Yaskawa INFORM job: A_ROOF_SIDE_0617_2_PAINT_47.JBI

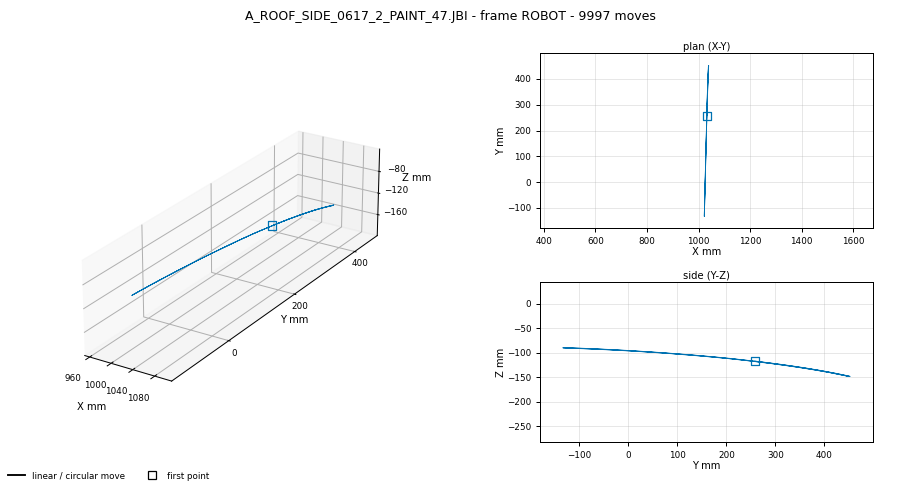
[picture p0: tool path of A_ROOF_SIDE_0617_2_PAINT_47.JBI in frame ROBOT, 9997 of 9997 moves have a stored position in this frame; points joined in program order, loops and branches not executed]
/JOB
//NAME A_ROOF_SIDE_0617_2_PAINT47
//POS
///NPOS 9997,0,0,0,0,0
///TOOL 1
///USER 0
///POSTYPE ROBOT
///RECTAN
///RCONF 1,0,0,0,0,0,0,0,0,0,0,0,0,0,0,0,0,0,0,0,0,0,0,0
C00000=1032.449,258.008,-117.083,170.684,44.569,158.533
C00001=1032.456,258.256,-117.113,170.687,44.569,158.534
C00002=1032.463,258.505,-117.142,170.690,44.569,158.534
C00003=1032.469,258.753,-117.172,170.693,44.568,158.534
C00004=1032.477,259.001,-117.201,170.697,44.568,158.535
C00005=1032.483,259.249,-117.230,170.701,44.568,158.535
C00006=1032.490,259.497,-117.260,170.704,44.568,158.535
C00007=1032.497,259.745,-117.290,170.707,44.567,158.535
C00008=1032.504,259.994,-117.319,170.711,44.567,158.536
C00009=1032.510,260.241,-117.349,170.714,44.567,158.536
C00010=1032.517,260.490,-117.379,170.718,44.567,158.536
C00011=1032.525,260.738,-117.408,170.721,44.567,158.537
C00012=1032.531,260.986,-117.437,170.725,44.566,158.537
C00013=1032.538,261.234,-117.467,170.728,44.566,158.537
C00014=1032.545,261.482,-117.497,170.731,44.566,158.537
C00015=1032.552,261.730,-117.527,170.734,44.566,158.538
C00016=1032.558,261.979,-117.556,170.739,44.566,158.538
C00017=1032.565,262.227,-117.586,170.742,44.566,158.538
C00018=1032.572,262.475,-117.617,170.745,44.566,158.539
C00019=1032.581,262.826,-117.659,170.749,44.566,158.539
C00020=1032.590,263.179,-117.701,170.755,44.566,158.540
C00021=1032.600,263.530,-117.744,170.759,44.566,158.540
C00022=1032.609,263.882,-117.786,170.765,44.566,158.541
C00023=1032.616,264.130,-117.817,170.768,44.566,158.541
C00024=1032.623,264.378,-117.846,170.771,44.566,158.541
C00025=1032.630,264.626,-117.876,170.775,44.566,158.541
C00026=1032.636,264.875,-117.907,170.779,44.566,158.542
C00027=1032.643,265.122,-117.937,170.782,44.566,158.542
C00028=1032.650,265.370,-117.967,170.786,44.566,158.542
C00029=1032.656,265.619,-117.997,170.789,44.566,158.543
C00030=1032.662,265.867,-118.027,170.792,44.566,158.543
C00031=1032.670,266.115,-118.057,170.796,44.565,158.543
C00032=1032.677,266.363,-118.087,170.800,44.565,158.544
C00033=1032.683,266.611,-118.117,170.803,44.565,158.544
C00034=1032.690,266.859,-118.148,170.806,44.565,158.544
C00035=1032.697,267.108,-118.178,170.810,44.565,158.545
C00036=1032.703,267.355,-118.208,170.814,44.565,158.545
C00037=1032.710,267.604,-118.238,170.817,44.565,158.545
C00038=1032.717,267.851,-118.269,170.821,44.566,158.546
C00039=1032.723,268.099,-118.299,170.824,44.566,158.546
C00040=1032.730,268.347,-118.329,170.828,44.565,158.546
C00041=1032.737,268.596,-118.360,170.831,44.565,158.547
C00042=1032.743,268.843,-118.390,170.835,44.565,158.547
C00043=1032.750,269.092,-118.421,170.838,44.565,158.547
C00044=1032.757,269.340,-118.451,170.842,44.566,158.548
C00045=1032.764,269.588,-118.481,170.846,44.566,158.548
C00046=1032.770,269.835,-118.512,170.849,44.566,158.549
C00047=1032.777,270.084,-118.542,170.852,44.566,158.549
C00048=1032.784,270.332,-118.573,170.856,44.566,158.549
C00049=1032.791,270.580,-118.603,170.860,44.566,158.549
C00050=1032.797,270.828,-118.634,170.864,44.566,158.550
C00051=1032.804,271.076,-118.664,170.867,44.566,158.550
C00052=1032.811,271.324,-118.695,170.870,44.566,158.551
C00053=1032.818,271.573,-118.725,170.874,44.566,158.551
C00054=1032.824,271.820,-118.756,170.878,44.567,158.551
C00055=1032.831,272.068,-118.786,170.881,44.566,158.552
C00056=1032.837,272.317,-118.817,170.885,44.566,158.552
C00057=1032.844,272.564,-118.848,170.889,44.567,158.553
C00058=1032.851,272.812,-118.878,170.892,44.567,158.553
C00059=1032.857,273.060,-118.909,170.896,44.567,158.553
C00060=1032.865,273.308,-118.940,170.900,44.567,158.554
C00061=1032.871,273.557,-118.970,170.903,44.567,158.554
C00062=1032.878,273.804,-119.002,170.907,44.567,158.554
C00063=1032.884,274.052,-119.031,170.910,44.568,158.555
C00064=1032.891,274.300,-119.063,170.914,44.568,158.555
C00065=1032.897,274.548,-119.094,170.918,44.568,158.555
C00066=1032.905,274.796,-119.124,170.921,44.568,158.556
C00067=1032.911,275.045,-119.155,170.926,44.568,158.556
C00068=1032.918,275.292,-119.187,170.929,44.568,158.557
C00069=1032.925,275.540,-119.216,170.932,44.569,158.557
C00070=1032.931,275.788,-119.248,170.936,44.569,158.557
C00071=1032.938,276.036,-119.279,170.940,44.569,158.558
C00072=1032.945,276.284,-119.309,170.943,44.569,158.558
C00073=1032.952,276.532,-119.341,170.947,44.569,158.558
C00074=1032.958,276.780,-119.372,170.951,44.569,158.559
C00075=1032.969,277.137,-119.415,170.957,44.569,158.560
C00076=1032.978,277.493,-119.460,170.961,44.570,158.560
C00077=1032.988,277.850,-119.505,170.967,44.570,158.561
C00078=1032.997,278.206,-119.549,170.972,44.570,158.561
C00079=1033.004,278.453,-119.581,170.976,44.571,158.562
C00080=1033.011,278.702,-119.612,170.980,44.571,158.562
C00081=1033.017,278.950,-119.643,170.984,44.571,158.562
C00082=1033.024,279.198,-119.674,170.987,44.571,158.563
C00083=1033.031,279.446,-119.706,170.992,44.572,158.563
C00084=1033.037,279.694,-119.737,170.995,44.572,158.564
C00085=1033.044,279.942,-119.768,170.998,44.572,158.564
C00086=1033.051,280.190,-119.799,171.003,44.573,158.565
C00087=1033.058,280.438,-119.830,171.006,44.573,158.565
C00088=1033.065,280.686,-119.862,171.010,44.573,158.565
C00089=1033.071,280.933,-119.893,171.014,44.573,158.566
C00090=1033.078,281.181,-119.925,171.018,44.574,158.566
C00091=1033.085,281.429,-119.956,171.021,44.574,158.567
C00092=1033.092,281.677,-119.987,171.025,44.574,158.567
C00093=1033.098,281.925,-120.019,171.029,44.575,158.568
C00094=1033.105,282.173,-120.050,171.032,44.575,158.568
C00095=1033.112,282.421,-120.082,171.037,44.575,158.568
C00096=1033.119,282.669,-120.113,171.040,44.576,158.569
C00097=1033.125,282.917,-120.145,171.045,44.575,158.569
C00098=1033.132,283.165,-120.176,171.048,44.576,158.570
C00099=1033.139,283.412,-120.207,171.052,44.577,158.570
C00100=1033.145,283.660,-120.239,171.056,44.576,158.570
C00101=1033.153,283.908,-120.270,171.059,44.577,158.571
C00102=1033.160,284.156,-120.301,171.064,44.577,158.571
C00103=1033.166,284.404,-120.333,171.067,44.578,158.572
C00104=1033.173,284.652,-120.364,171.071,44.578,158.572
C00105=1033.180,284.900,-120.395,171.075,44.578,158.573
C00106=1033.187,285.147,-120.427,171.079,44.579,158.573
C00107=1033.194,285.396,-120.459,171.083,44.579,158.574
C00108=1033.201,285.644,-120.490,171.087,44.579,158.574
C00109=1033.208,285.891,-120.522,171.091,44.580,158.575
C00110=1033.214,286.139,-120.554,171.094,44.580,158.575
C00111=1033.221,286.387,-120.585,171.098,44.580,158.575
C00112=1033.228,286.635,-120.617,171.102,44.581,158.576
C00113=1033.235,286.883,-120.648,171.106,44.581,158.576
C00114=1033.241,287.130,-120.681,171.111,44.582,158.577
C00115=1033.248,287.379,-120.713,171.114,44.582,158.577
C00116=1033.255,287.627,-120.744,171.118,44.582,158.578
C00117=1033.262,287.874,-120.776,171.122,44.583,158.578
C00118=1033.269,288.122,-120.808,171.125,44.583,158.579
C00119=1033.275,288.370,-120.839,171.130,44.584,158.579
C00120=1033.282,288.618,-120.872,171.133,44.584,158.580
C00121=1033.289,288.866,-120.904,171.138,44.585,158.580
C00122=1033.296,289.114,-120.936,171.142,44.585,158.581
C00123=1033.303,289.361,-120.967,171.146,44.585,158.581
C00124=1033.310,289.609,-120.999,171.150,44.586,158.582
C00125=1033.316,289.857,-121.031,171.154,44.586,158.582
C00126=1033.322,290.105,-121.063,171.157,44.586,158.582
C00127=1033.330,290.353,-121.095,171.162,44.587,158.583
C00128=1033.337,290.601,-121.127,171.165,44.587,158.583
C00129=1033.343,290.848,-121.159,171.170,44.588,158.584
C00130=1033.350,291.096,-121.192,171.174,44.588,158.584
C00131=1033.361,291.464,-121.239,171.179,44.589,158.585
C00132=1033.371,291.833,-121.287,171.185,44.590,158.586
C00133=1033.381,292.202,-121.335,171.192,44.591,158.587
C00134=1033.391,292.570,-121.383,171.198,44.591,158.587
C00135=1033.398,292.818,-121.414,171.201,44.592,158.588
C00136=1033.405,293.066,-121.447,171.206,44.592,158.588
C00137=1033.412,293.314,-121.479,171.209,44.593,158.589
C00138=1033.418,293.561,-121.511,171.214,44.593,158.589
C00139=1033.425,293.810,-121.544,171.218,44.595,158.590
C00140=1033.432,294.057,-121.576,171.222,44.595,158.590
C00141=1033.439,294.304,-121.608,171.226,44.596,158.591
C00142=1033.446,294.553,-121.641,171.230,44.596,158.591
C00143=1033.453,294.801,-121.673,171.234,44.596,158.592
C00144=1033.459,295.048,-121.705,171.238,44.597,158.592
C00145=1033.466,295.296,-121.738,171.242,44.598,158.593
C00146=1033.473,295.544,-121.771,171.247,44.598,158.594
C00147=1033.479,295.791,-121.803,171.250,44.599,158.594
C00148=1033.486,296.039,-121.836,171.255,44.599,158.595
C00149=1033.493,296.287,-121.869,171.258,44.601,158.595
C00150=1033.500,296.534,-121.901,171.263,44.601,158.596
C00151=1033.506,296.782,-121.934,171.267,44.601,158.596
C00152=1033.513,297.030,-121.967,171.271,44.603,158.597
C00153=1033.520,297.278,-121.999,171.276,44.603,158.597
C00154=1033.526,297.525,-122.032,171.279,44.604,158.598
C00155=1033.533,297.774,-122.065,171.284,44.605,158.599
C00156=1033.540,298.021,-122.097,171.288,44.605,158.599
C00157=1033.546,298.268,-122.130,171.292,44.606,158.600
C00158=1033.553,298.517,-122.163,171.296,44.607,158.600
C00159=1033.560,298.764,-122.197,171.300,44.607,158.601
C00160=1033.568,299.012,-122.229,171.304,44.608,158.601
C00161=1033.574,299.259,-122.262,171.309,44.609,158.602
C00162=1033.580,299.507,-122.295,171.313,44.609,158.602
C00163=1033.587,299.755,-122.328,171.317,44.610,158.603
C00164=1033.594,300.002,-122.360,171.322,44.611,158.603
C00165=1033.601,300.250,-122.394,171.325,44.612,158.604
C00166=1033.608,300.498,-122.427,171.330,44.612,158.605
C00167=1033.615,300.746,-122.459,171.334,44.613,158.605
C00168=1033.621,300.993,-122.492,171.338,44.614,158.606
C00169=1033.629,301.241,-122.526,171.343,44.614,158.606
C00170=1033.635,301.489,-122.558,171.347,44.615,158.607
C00171=1033.643,301.737,-122.591,171.351,44.616,158.607
C00172=1033.649,301.983,-122.624,171.356,44.617,158.608
C00173=1033.656,302.232,-122.657,171.359,44.617,158.609
C00174=1033.662,302.479,-122.690,171.364,44.618,158.609
C00175=1033.670,302.727,-122.723,171.368,44.619,158.610
C00176=1033.677,302.974,-122.756,171.373,44.620,158.610
C00177=1033.684,303.223,-122.789,171.377,44.620,158.611
C00178=1033.690,303.470,-122.823,171.381,44.622,158.612
C00179=1033.698,303.718,-122.855,171.385,44.622,158.612
C00180=1033.705,303.965,-122.889,171.390,44.623,158.613
C00181=1033.711,304.213,-122.922,171.394,44.623,158.613
C00182=1033.718,304.461,-122.956,171.399,44.624,158.614
C00183=1033.725,304.708,-122.988,171.403,44.625,158.614
C00184=1033.733,304.955,-123.022,171.407,44.626,158.615
C00185=1033.740,305.204,-123.055,171.412,44.627,158.616
C00186=1033.746,305.451,-123.088,171.416,44.627,158.616
C00187=1033.757,305.836,-123.139,171.422,44.629,158.617
C00188=1033.768,306.222,-123.192,171.429,44.630,158.618
C00189=1033.779,306.608,-123.243,171.436,44.631,158.619
C00190=1033.791,306.993,-123.295,171.443,44.632,158.620
C00191=1033.798,307.241,-123.328,171.448,44.633,158.621
C00192=1033.804,307.488,-123.362,171.452,44.634,158.621
C00193=1033.811,307.736,-123.395,171.456,44.635,158.622
C00194=1033.818,307.984,-123.428,171.461,44.636,158.623
C00195=1033.826,308.231,-123.462,171.465,44.637,158.623
C00196=1033.833,308.478,-123.495,171.470,44.638,158.624
C00197=1033.840,308.726,-123.529,171.474,44.638,158.624
C00198=1033.847,308.974,-123.562,171.479,44.639,158.625
C00199=1033.855,309.222,-123.595,171.483,44.641,158.626
C00200=1033.861,309.469,-123.629,171.487,44.641,158.626
C00201=1033.869,309.716,-123.663,171.492,44.642,158.627
C00202=1033.876,309.964,-123.696,171.497,44.643,158.628
C00203=1033.883,310.212,-123.730,171.502,44.644,158.628
C00204=1033.891,310.460,-123.763,171.505,44.644,158.629
C00205=1033.898,310.707,-123.797,171.510,44.645,158.629
C00206=1033.904,310.954,-123.830,171.515,44.646,158.630
C00207=1033.912,311.202,-123.864,171.520,44.647,158.631
C00208=1033.919,311.450,-123.898,171.524,44.648,158.631
C00209=1033.926,311.697,-123.932,171.528,44.650,158.632
C00210=1033.933,311.945,-123.965,171.533,44.651,158.633
C00211=1033.939,312.192,-123.999,171.538,44.651,158.633
C00212=1033.946,312.440,-124.033,171.542,44.653,158.634
C00213=1033.953,312.688,-124.067,171.546,44.654,158.635
C00214=1033.960,312.935,-124.102,171.551,44.655,158.635
C00215=1033.967,313.183,-124.136,171.556,44.656,158.636
C00216=1033.973,313.430,-124.170,171.560,44.657,158.637
C00217=1033.981,313.678,-124.204,171.565,44.658,158.637
C00218=1033.988,313.925,-124.238,171.569,44.659,158.638
C00219=1033.994,314.173,-124.273,171.574,44.660,158.639
C00220=1034.002,314.420,-124.307,171.579,44.661,158.640
C00221=1034.008,314.668,-124.341,171.583,44.663,158.640
C00222=1034.016,314.915,-124.376,171.588,44.663,158.641
C00223=1034.022,315.162,-124.409,171.593,44.664,158.642
C00224=1034.029,315.410,-124.444,171.597,44.665,158.642
C00225=1034.036,315.657,-124.478,171.602,44.667,158.643
C00226=1034.043,315.905,-124.512,171.606,44.668,158.644
C00227=1034.050,316.152,-124.547,171.611,44.669,158.645
C00228=1034.057,316.400,-124.581,171.616,44.670,158.645
C00229=1034.064,316.648,-124.615,171.621,44.671,158.646
C00230=1034.071,316.895,-124.650,171.626,44.673,158.647
C00231=1034.078,317.143,-124.684,171.629,44.674,158.647
C00232=1034.085,317.390,-124.719,171.634,44.675,158.648
C00233=1034.092,317.638,-124.753,171.639,44.676,158.649
C00234=1034.099,317.885,-124.788,171.644,44.677,158.650
C00235=1034.106,318.133,-124.822,171.649,44.678,158.650
C00236=1034.113,318.380,-124.857,171.654,44.679,158.651
C00237=1034.120,318.628,-124.890,171.659,44.681,158.652
C00238=1034.127,318.875,-124.926,171.662,44.682,158.652
C00239=1034.135,319.122,-124.960,171.667,44.683,158.653
C00240=1034.141,319.370,-124.995,171.672,44.685,158.654
C00241=1034.149,319.617,-125.029,171.677,44.686,158.655
C00242=1034.157,319.866,-125.063,171.682,44.687,158.655
C00243=1034.167,320.256,-125.118,171.689,44.689,158.657
C00244=1034.179,320.646,-125.173,171.697,44.691,158.658
C00245=1034.189,321.036,-125.227,171.705,44.692,158.659
C00246=1034.201,321.427,-125.282,171.713,44.695,158.660
C00247=1034.209,321.674,-125.317,171.717,44.696,158.661
C00248=1034.215,321.922,-125.351,171.722,44.697,158.662
C00249=1034.223,322.169,-125.386,171.727,44.698,158.662
C00250=1034.230,322.417,-125.421,171.731,44.700,158.663
C00251=1034.238,322.664,-125.456,171.736,44.701,158.664
C00252=1034.244,322.911,-125.491,171.741,44.702,158.665
C00253=1034.252,323.158,-125.525,171.746,44.703,158.665
C00254=1034.259,323.407,-125.560,171.751,44.705,158.666
C00255=1034.266,323.654,-125.595,171.756,44.706,158.667
C00256=1034.273,323.901,-125.630,171.761,44.707,158.668
C00257=1034.281,324.149,-125.665,171.766,44.708,158.669
C00258=1034.288,324.396,-125.700,171.771,44.710,158.669
C00259=1034.296,324.643,-125.735,171.775,44.711,158.670
C00260=1034.303,324.892,-125.770,171.780,44.712,158.671
C00261=1034.310,325.139,-125.805,171.785,44.714,158.672
C00262=1034.317,325.386,-125.840,171.790,44.715,158.672
C00263=1034.325,325.634,-125.875,171.795,44.717,158.673
C00264=1034.332,325.881,-125.910,171.800,44.718,158.674
C00265=1034.340,326.128,-125.944,171.805,44.719,158.675
C00266=1034.347,326.376,-125.980,171.810,44.721,158.676
C00267=1034.354,326.623,-126.014,171.815,44.722,158.676
C00268=1034.362,326.870,-126.050,171.820,44.723,158.677
C00269=1034.370,327.118,-126.085,171.826,44.724,158.678
C00270=1034.376,327.365,-126.120,171.831,44.726,158.679
C00271=1034.385,327.613,-126.155,171.836,44.727,158.680
C00272=1034.391,327.860,-126.190,171.841,44.729,158.681
C00273=1034.399,328.108,-126.225,171.846,44.730,158.681
C00274=1034.406,328.355,-126.261,171.851,44.732,158.682
C00275=1034.414,328.603,-126.297,171.856,44.733,158.683
C00276=1034.421,328.850,-126.332,171.861,44.734,158.684
C00277=1034.428,329.097,-126.367,171.866,44.736,158.685
C00278=1034.436,329.345,-126.402,171.871,44.737,158.686
C00279=1034.443,329.591,-126.438,171.876,44.739,158.686
C00280=1034.450,329.839,-126.474,171.881,44.740,158.687
C00281=1034.457,330.086,-126.510,171.886,44.742,158.688
C00282=1034.465,330.334,-126.545,171.891,44.744,158.689
C00283=1034.472,330.581,-126.581,171.896,44.745,158.690
C00284=1034.479,330.829,-126.616,171.901,44.747,158.691
C00285=1034.486,331.076,-126.652,171.906,44.748,158.691
C00286=1034.494,331.324,-126.688,171.912,44.750,158.692
C00287=1034.501,331.571,-126.724,171.917,44.751,158.693
C00288=1034.508,331.818,-126.760,171.922,44.753,158.694
C00289=1034.515,332.065,-126.795,171.928,44.755,158.695
C00290=1034.524,332.313,-126.831,171.933,44.756,158.696
C00291=1034.530,332.560,-126.866,171.938,44.758,158.697
C00292=1034.538,332.807,-126.902,171.943,44.759,158.698
C00293=1034.546,333.055,-126.938,171.948,44.761,158.699
C00294=1034.553,333.302,-126.974,171.954,44.762,158.699
C00295=1034.560,333.550,-127.010,171.959,44.764,158.700
C00296=1034.567,333.796,-127.045,171.964,44.766,158.701
C00297=1034.575,334.044,-127.082,171.969,44.768,158.702
C00298=1034.583,334.291,-127.118,171.974,44.769,158.703
C00299=1034.594,334.678,-127.174,171.983,44.772,158.705
C00300=1034.605,335.063,-127.230,171.991,44.774,158.706
C00301=1034.617,335.448,-127.286,172.000,44.777,158.707
C00302=1034.628,335.834,-127.343,172.008,44.780,158.709
C00303=1034.635,336.082,-127.380,172.013,44.781,158.710
C00304=1034.642,336.329,-127.415,172.018,44.783,158.711
C00305=1034.650,336.576,-127.452,172.024,44.785,158.712
C00306=1034.658,336.823,-127.488,172.029,44.786,158.712
C00307=1034.665,337.070,-127.524,172.034,44.788,158.713
C00308=1034.672,337.318,-127.561,172.039,44.790,158.714
C00309=1034.679,337.565,-127.597,172.045,44.792,158.715
C00310=1034.687,337.813,-127.633,172.051,44.793,158.716
C00311=1034.695,338.060,-127.670,172.056,44.796,158.717
C00312=1034.702,338.306,-127.706,172.061,44.797,158.718
C00313=1034.709,338.554,-127.743,172.066,44.799,158.719
C00314=1034.717,338.802,-127.779,172.073,44.801,158.720
C00315=1034.724,339.049,-127.815,172.078,44.803,158.721
C00316=1034.732,339.296,-127.852,172.083,44.804,158.722
C00317=1034.740,339.543,-127.888,172.088,44.806,158.723
C00318=1034.746,339.790,-127.925,172.095,44.808,158.724
C00319=1034.754,340.037,-127.962,172.100,44.810,158.725
C00320=1034.762,340.285,-127.998,172.105,44.812,158.726
C00321=1034.770,340.532,-128.034,172.111,44.813,158.727
C00322=1034.778,340.779,-128.071,172.116,44.815,158.728
C00323=1034.785,341.027,-128.108,172.122,44.818,158.729
C00324=1034.793,341.273,-128.145,172.127,44.820,158.730
C00325=1034.799,341.521,-128.181,172.133,44.821,158.731
C00326=1034.807,341.767,-128.218,172.138,44.823,158.732
C00327=1034.815,342.015,-128.254,172.144,44.825,158.733
C00328=1034.822,342.262,-128.292,172.150,44.827,158.734
C00329=1034.830,342.509,-128.328,172.155,44.829,158.735
C00330=1034.837,342.756,-128.366,172.160,44.831,158.736
C00331=1034.845,343.003,-128.402,172.167,44.833,158.737
C00332=1034.852,343.251,-128.439,172.172,44.835,158.738
C00333=1034.860,343.498,-128.476,172.177,44.837,158.739
C00334=1034.867,343.745,-128.514,172.184,44.839,158.740
C00335=1034.875,343.992,-128.550,172.189,44.841,158.741
C00336=1034.882,344.240,-128.587,172.194,44.843,158.742
C00337=1034.890,344.486,-128.624,172.200,44.845,158.743
C00338=1034.897,344.734,-128.662,172.206,44.847,158.744
C00339=1034.905,344.981,-128.698,172.211,44.849,158.745
C00340=1034.912,345.228,-128.736,172.217,44.851,158.746
C00341=1034.920,345.475,-128.773,172.223,44.853,158.747
C00342=1034.927,345.722,-128.810,172.228,44.855,158.748
C00343=1034.935,345.969,-128.847,172.234,44.857,158.749
C00344=1034.942,346.216,-128.885,172.240,44.859,158.750
C00345=1034.951,346.464,-128.922,172.246,44.861,158.752
C00346=1034.958,346.711,-128.959,172.251,44.863,158.753
C00347=1034.966,346.958,-128.997,172.257,44.866,158.754
C00348=1034.974,347.205,-129.034,172.263,44.867,158.755
C00349=1034.981,347.452,-129.071,172.269,44.870,158.756
C00350=1034.989,347.699,-129.108,172.275,44.872,158.757
C00351=1034.997,347.946,-129.146,172.280,44.874,158.758
C00352=1035.005,348.193,-129.183,172.287,44.876,158.759
C00353=1035.012,348.440,-129.221,172.292,44.878,158.760
C00354=1035.019,348.688,-129.258,172.298,44.881,158.761
C00355=1035.032,349.070,-129.316,172.308,44.884,158.763
C00356=1035.043,349.452,-129.375,172.316,44.887,158.765
C00357=1035.055,349.835,-129.432,172.325,44.891,158.766
C00358=1035.067,350.217,-129.491,172.334,44.894,158.768
C00359=1035.075,350.464,-129.529,172.341,44.896,158.769
C00360=1035.082,350.711,-129.566,172.346,44.899,158.771
C00361=1035.090,350.957,-129.604,172.352,44.901,158.772
C00362=1035.098,351.205,-129.642,172.358,44.904,158.773
C00363=1035.105,351.452,-129.680,172.364,44.905,158.774
C00364=1035.113,351.699,-129.718,172.370,44.908,158.775
C00365=1035.121,351.946,-129.756,172.376,44.910,158.776
C00366=1035.128,352.193,-129.794,172.382,44.913,158.777
C00367=1035.136,352.440,-129.832,172.388,44.915,158.778
C00368=1035.144,352.687,-129.869,172.395,44.917,158.780
C00369=1035.152,352.934,-129.908,172.400,44.920,158.781
C00370=1035.159,353.180,-129.946,172.407,44.922,158.782
C00371=1035.167,353.428,-129.984,172.412,44.924,158.783
C00372=1035.175,353.675,-130.022,172.419,44.926,158.784
C00373=1035.184,353.922,-130.060,172.424,44.929,158.785
C00374=1035.191,354.169,-130.098,172.431,44.931,158.787
C00375=1035.199,354.416,-130.136,172.437,44.934,158.788
C00376=1035.207,354.663,-130.174,172.443,44.936,158.789
C00377=1035.214,354.910,-130.212,172.449,44.938,158.790
C00378=1035.222,355.157,-130.251,172.455,44.941,158.791
C00379=1035.230,355.404,-130.289,172.461,44.944,158.793
C00380=1035.238,355.650,-130.327,172.468,44.945,158.794
C00381=1035.247,355.898,-130.365,172.473,44.948,158.795
C00382=1035.254,356.144,-130.404,172.480,44.951,158.796
C00383=1035.262,356.391,-130.442,172.487,44.953,158.798
C00384=1035.270,356.638,-130.481,172.492,44.956,158.799
C00385=1035.277,356.885,-130.520,172.499,44.958,158.800
C00386=1035.285,357.132,-130.558,172.505,44.961,158.801
C00387=1035.293,357.379,-130.597,172.511,44.963,158.802
C00388=1035.301,357.626,-130.635,172.518,44.966,158.804
C00389=1035.309,357.873,-130.673,172.524,44.968,158.805
C00390=1035.317,358.120,-130.712,172.530,44.971,158.806
C00391=1035.324,358.366,-130.750,172.536,44.973,158.807
C00392=1035.333,358.614,-130.789,172.543,44.976,158.809
C00393=1035.341,358.861,-130.828,172.549,44.978,158.810
C00394=1035.349,359.107,-130.867,172.555,44.981,158.811
C00395=1035.357,359.354,-130.905,172.562,44.983,158.812
C00396=1035.365,359.601,-130.944,172.569,44.986,158.814
C00397=1035.372,359.848,-130.982,172.574,44.989,158.815
C00398=1035.381,360.094,-131.021,172.581,44.992,158.816
C00399=1035.389,360.342,-131.060,172.587,44.994,158.818
C00400=1035.396,360.588,-131.099,172.594,44.997,158.819
C00401=1035.404,360.835,-131.138,172.600,45.000,158.820
C00402=1035.412,361.082,-131.177,172.606,45.002,158.821
C00403=1035.421,361.329,-131.216,172.613,45.005,158.823
C00404=1035.428,361.575,-131.254,172.620,45.008,158.824
C00405=1035.436,361.822,-131.294,172.627,45.010,158.825
C00406=1035.444,362.069,-131.333,172.632,45.013,158.827
C00407=1035.453,362.316,-131.372,172.639,45.016,158.828
C00408=1035.460,362.563,-131.412,172.646,45.019,158.830
C00409=1035.468,362.809,-131.450,172.652,45.021,158.831
C00410=1035.476,363.056,-131.490,172.659,45.024,158.832
C00411=1035.488,363.445,-131.552,172.669,45.029,158.834
C00412=1035.502,363.833,-131.614,172.680,45.033,158.836
C00413=1035.514,364.222,-131.675,172.690,45.038,158.839
C00414=1035.527,364.610,-131.738,172.700,45.042,158.841
C00415=1035.534,364.857,-131.778,172.707,45.045,158.842
C00416=1035.543,365.104,-131.816,172.714,45.048,158.844
C00417=1035.551,365.351,-131.856,172.721,45.050,158.845
C00418=1035.559,365.597,-131.895,172.728,45.053,158.846
C00419=1035.567,365.844,-131.935,172.734,45.056,158.848
C00420=1035.575,366.091,-131.975,172.741,45.059,158.849
C00421=1035.583,366.338,-132.014,172.747,45.062,158.850
C00422=1035.592,366.584,-132.053,172.754,45.065,158.852
C00423=1035.600,366.831,-132.093,172.761,45.068,158.853
C00424=1035.608,367.078,-132.133,172.768,45.071,158.855
C00425=1035.616,367.324,-132.173,172.774,45.074,158.856
C00426=1035.625,367.570,-132.213,172.781,45.077,158.858
C00427=1035.633,367.817,-132.252,172.788,45.080,158.859
C00428=1035.641,368.064,-132.292,172.795,45.083,158.860
C00429=1035.649,368.311,-132.331,172.802,45.086,158.862
C00430=1035.658,368.558,-132.372,172.809,45.089,158.863
C00431=1035.666,368.804,-132.411,172.816,45.092,158.865
C00432=1035.675,369.051,-132.451,172.823,45.095,158.866
C00433=1035.682,369.298,-132.491,172.829,45.098,158.868
C00434=1035.691,369.544,-132.531,172.836,45.101,158.869
C00435=1035.699,369.791,-132.571,172.843,45.104,158.870
C00436=1035.708,370.037,-132.611,172.850,45.107,158.872
C00437=1035.716,370.284,-132.651,172.857,45.110,158.873
C00438=1035.724,370.530,-132.692,172.864,45.113,158.875
C00439=1035.732,370.777,-132.732,172.872,45.116,158.876
C00440=1035.741,371.023,-132.772,172.879,45.119,158.878
C00441=1035.748,371.270,-132.811,172.886,45.123,158.880
C00442=1035.757,371.517,-132.853,172.893,45.126,158.881
C00443=1035.765,371.763,-132.893,172.900,45.129,158.882
C00444=1035.773,372.010,-132.932,172.907,45.132,158.884
C00445=1035.781,372.256,-132.973,172.914,45.135,158.885
C00446=1035.790,372.503,-133.014,172.921,45.139,158.887
C00447=1035.798,372.750,-133.055,172.928,45.142,158.889
C00448=1035.807,372.996,-133.095,172.935,45.145,158.890
C00449=1035.815,373.243,-133.135,172.943,45.148,158.892
C00450=1035.823,373.489,-133.176,172.950,45.152,158.893
C00451=1035.831,373.736,-133.216,172.957,45.155,158.895
C00452=1035.841,373.982,-133.257,172.964,45.158,158.896
C00453=1035.849,374.229,-133.297,172.971,45.162,158.898
C00454=1035.857,374.476,-133.338,172.978,45.165,158.899
C00455=1035.865,374.722,-133.379,172.986,45.168,158.901
C00456=1035.874,374.968,-133.419,172.994,45.172,158.903
C00457=1035.883,375.215,-133.460,173.001,45.175,158.904
C00458=1035.891,375.461,-133.501,173.008,45.178,158.906
C00459=1035.899,375.708,-133.542,173.015,45.182,158.907
C00460=1035.908,375.954,-133.582,173.023,45.185,158.909
C00461=1035.917,376.201,-133.623,173.030,45.188,158.911
C00462=1035.925,376.447,-133.664,173.037,45.192,158.912
C00463=1035.934,376.694,-133.705,173.045,45.195,158.914
C00464=1035.942,376.940,-133.746,173.052,45.198,158.915
C00465=1035.951,377.187,-133.786,173.060,45.202,158.917
C00466=1035.960,377.433,-133.828,173.067,45.205,158.919
C00467=1035.974,377.842,-133.895,173.079,45.211,158.921
C00468=1035.988,378.251,-133.964,173.092,45.217,158.924
C00469=1036.002,378.660,-134.032,173.105,45.223,158.927
C00470=1036.016,379.069,-134.100,173.117,45.229,158.930
C00471=1036.025,379.315,-134.142,173.125,45.232,158.931
C00472=1036.033,379.562,-134.183,173.132,45.236,158.933
C00473=1036.041,379.808,-134.225,173.140,45.239,158.935
C00474=1036.050,380.055,-134.267,173.147,45.243,158.937
C00475=1036.059,380.300,-134.308,173.156,45.247,158.938
C00476=1036.067,380.547,-134.349,173.163,45.250,158.940
C00477=1036.076,380.794,-134.391,173.170,45.254,158.942
C00478=1036.085,381.040,-134.433,173.178,45.257,158.943
C00479=1036.094,381.286,-134.474,173.186,45.262,158.945
C00480=1036.102,381.532,-134.516,173.194,45.265,158.947
C00481=1036.111,381.779,-134.558,173.202,45.269,158.949
C00482=1036.119,382.026,-134.599,173.210,45.272,158.950
C00483=1036.128,382.272,-134.641,173.217,45.276,158.952
C00484=1036.137,382.518,-134.682,173.224,45.280,158.954
C00485=1036.146,382.764,-134.724,173.233,45.284,158.956
C00486=1036.154,383.010,-134.766,173.240,45.287,158.957
C00487=1036.164,383.256,-134.808,173.248,45.291,158.959
C00488=1036.173,383.503,-134.850,173.257,45.295,158.961
C00489=1036.181,383.749,-134.892,173.264,45.298,158.963
C00490=1036.190,383.996,-134.934,173.273,45.302,158.964
C00491=1036.199,384.242,-134.975,173.280,45.306,158.966
C00492=1036.208,384.488,-135.017,173.289,45.310,158.968
C00493=1036.217,384.734,-135.060,173.296,45.314,158.970
C00494=1036.226,384.980,-135.101,173.304,45.317,158.972
C00495=1036.235,385.227,-135.143,173.312,45.322,158.973
C00496=1036.243,385.473,-135.186,173.320,45.325,158.975
C00497=1036.252,385.719,-135.228,173.329,45.329,158.977
C00498=1036.261,385.966,-135.269,173.336,45.333,158.979
C00499=1036.270,386.211,-135.312,173.345,45.337,158.981
C00500=1036.279,386.458,-135.354,173.353,45.341,158.983
C00501=1036.289,386.703,-135.396,173.360,45.345,158.985
C00502=1036.297,386.950,-135.438,173.369,45.349,158.986
C00503=1036.306,387.196,-135.481,173.377,45.353,158.988
C00504=1036.315,387.443,-135.523,173.385,45.357,158.990
C00505=1036.325,387.689,-135.565,173.394,45.361,158.992
C00506=1036.333,387.935,-135.608,173.402,45.365,158.994
C00507=1036.342,388.181,-135.650,173.410,45.369,158.996
C00508=1036.351,388.427,-135.692,173.418,45.373,158.998
C00509=1036.360,388.673,-135.736,173.427,45.377,159.000
C00510=1036.370,388.919,-135.778,173.435,45.381,159.002
C00511=1036.378,389.165,-135.821,173.443,45.386,159.004
C00512=1036.387,389.411,-135.864,173.452,45.389,159.006
C00513=1036.396,389.657,-135.907,173.460,45.394,159.008
C00514=1036.406,389.904,-135.950,173.469,45.398,159.009
C00515=1036.415,390.149,-135.992,173.478,45.402,159.012
C00516=1036.424,390.395,-136.035,173.485,45.406,159.013
C00517=1036.433,390.642,-136.078,173.494,45.410,159.015
C00518=1036.442,390.888,-136.121,173.503,45.415,159.017
C00519=1036.451,391.134,-136.163,173.511,45.419,159.019
C00520=1036.460,391.380,-136.207,173.520,45.423,159.021
C00521=1036.469,391.626,-136.250,173.529,45.427,159.023
C00522=1036.478,391.872,-136.293,173.536,45.432,159.025
C00523=1036.489,392.155,-136.342,173.546,45.437,159.028
C00524=1036.499,392.436,-136.392,173.556,45.441,159.030
C00525=1036.509,392.719,-136.441,173.567,45.447,159.032
C00526=1036.521,393.001,-136.491,173.576,45.452,159.035
C00527=1036.530,393.246,-136.535,173.585,45.456,159.037
C00528=1036.539,393.493,-136.578,173.593,45.460,159.039
C00529=1036.548,393.738,-136.621,173.602,45.465,159.041
C00530=1036.557,393.985,-136.665,173.611,45.469,159.043
C00531=1036.573,394.392,-136.737,173.626,45.476,159.046
C00532=1036.588,394.800,-136.808,173.640,45.484,159.050
C00533=1036.604,395.207,-136.881,173.655,45.491,159.053
C00534=1036.619,395.614,-136.953,173.670,45.499,159.057
C00535=1036.629,395.860,-136.997,173.679,45.503,159.059
C00536=1036.638,396.106,-137.041,173.688,45.508,159.061
C00537=1036.647,396.352,-137.085,173.697,45.512,159.063
C00538=1036.657,396.597,-137.128,173.706,45.517,159.066
C00539=1036.666,396.844,-137.172,173.715,45.521,159.068
C00540=1036.675,397.089,-137.216,173.724,45.526,159.070
C00541=1036.685,397.335,-137.260,173.733,45.530,159.072
C00542=1036.694,397.581,-137.304,173.742,45.535,159.074
C00543=1036.704,397.827,-137.348,173.751,45.540,159.076
C00544=1036.714,398.073,-137.392,173.760,45.544,159.079
C00545=1036.722,398.319,-137.436,173.769,45.549,159.081
C00546=1036.732,398.564,-137.480,173.779,45.554,159.083
C00547=1036.741,398.810,-137.524,173.788,45.558,159.085
C00548=1036.752,399.056,-137.568,173.797,45.563,159.087
C00549=1036.761,399.302,-137.612,173.806,45.568,159.090
C00550=1036.771,399.548,-137.657,173.816,45.573,159.092
C00551=1036.780,399.794,-137.701,173.826,45.577,159.094
C00552=1036.790,400.039,-137.746,173.835,45.582,159.097
C00553=1036.799,400.286,-137.790,173.844,45.587,159.099
C00554=1036.809,400.531,-137.835,173.854,45.592,159.101
C00555=1036.818,400.777,-137.879,173.863,45.597,159.103
C00556=1036.828,401.023,-137.924,173.872,45.602,159.106
C00557=1036.837,401.269,-137.968,173.882,45.606,159.108
C00558=1036.847,401.514,-138.013,173.891,45.612,159.110
C00559=1036.857,401.760,-138.057,173.901,45.616,159.113
C00560=1036.867,402.005,-138.102,173.911,45.621,159.115
C00561=1036.876,402.252,-138.146,173.920,45.626,159.117
C00562=1036.886,402.497,-138.191,173.930,45.631,159.120
C00563=1036.896,402.743,-138.236,173.939,45.636,159.122
C00564=1036.906,402.989,-138.281,173.949,45.641,159.124
C00565=1036.916,403.234,-138.326,173.959,45.646,159.127
C00566=1036.924,403.480,-138.372,173.968,45.651,159.129
C00567=1036.934,403.726,-138.416,173.978,45.656,159.132
C00568=1036.945,403.972,-138.462,173.988,45.661,159.134
C00569=1036.954,404.217,-138.506,173.998,45.666,159.136
C00570=1036.964,404.463,-138.551,174.007,45.672,159.139
C00571=1036.973,404.708,-138.597,174.018,45.677,159.141
C00572=1036.984,404.954,-138.642,174.027,45.682,159.144
C00573=1036.993,405.200,-138.687,174.037,45.687,159.146
C00574=1037.003,405.445,-138.733,174.047,45.692,159.149
C00575=1037.013,405.691,-138.779,174.057,45.697,159.151
C00576=1037.023,405.937,-138.823,174.066,45.703,159.154
C00577=1037.033,406.182,-138.869,174.077,45.708,159.156
C00578=1037.043,406.428,-138.914,174.087,45.713,159.159
C00579=1037.053,406.660,-138.957,174.097,45.718,159.161
C00580=1037.061,406.892,-139.000,174.106,45.723,159.163
C00581=1037.071,407.123,-139.044,174.116,45.728,159.166
C00582=1037.080,407.356,-139.087,174.125,45.733,159.168
C00583=1037.090,407.588,-139.130,174.135,45.738,159.171
C00584=1037.099,407.820,-139.173,174.144,45.743,159.173
C00585=1037.110,408.051,-139.216,174.154,45.748,159.175
C00586=1037.118,408.283,-139.259,174.164,45.754,159.178
C00587=1037.129,408.528,-139.305,174.174,45.759,159.180
C00588=1037.139,408.775,-139.351,174.185,45.764,159.183
C00589=1037.149,409.020,-139.396,174.195,45.769,159.185
C00590=1037.159,409.265,-139.442,174.205,45.775,159.188
C00591=1037.169,409.511,-139.489,174.215,45.780,159.191
C00592=1037.179,409.756,-139.534,174.226,45.786,159.193
C00593=1037.190,410.002,-139.580,174.237,45.791,159.196
C00594=1037.200,410.247,-139.626,174.247,45.797,159.199
C00595=1037.210,410.493,-139.673,174.258,45.802,159.201
C00596=1037.221,410.739,-139.718,174.269,45.808,159.204
C00597=1037.232,410.985,-139.764,174.279,45.814,159.207
C00598=1037.241,411.229,-139.811,174.289,45.819,159.209
C00599=1037.252,411.475,-139.857,174.300,45.824,159.212
C00600=1037.262,411.721,-139.904,174.310,45.830,159.215
C00601=1037.273,411.966,-139.950,174.321,45.836,159.217
C00602=1037.283,412.211,-139.997,174.332,45.842,159.220
C00603=1037.293,412.457,-140.044,174.343,45.847,159.223
C00604=1037.303,412.702,-140.090,174.354,45.853,159.226
C00605=1037.314,412.948,-140.137,174.364,45.859,159.228
C00606=1037.324,413.193,-140.183,174.375,45.865,159.231
C00607=1037.334,413.439,-140.230,174.387,45.870,159.234
C00608=1037.345,413.684,-140.277,174.398,45.876,159.237
C00609=1037.355,413.929,-140.323,174.409,45.882,159.240
C00610=1037.365,414.175,-140.371,174.420,45.887,159.242
C00611=1037.376,414.420,-140.417,174.431,45.894,159.245
C00612=1037.386,414.665,-140.464,174.442,45.900,159.248
C00613=1037.397,414.911,-140.512,174.452,45.905,159.251
C00614=1037.408,415.156,-140.559,174.464,45.911,159.254
C00615=1037.418,415.401,-140.606,174.476,45.917,159.257
C00616=1037.429,415.646,-140.653,174.486,45.923,159.259
C00617=1037.439,415.891,-140.700,174.497,45.929,159.262
C00618=1037.450,416.137,-140.747,174.509,45.935,159.265
C00619=1037.461,416.382,-140.794,174.520,45.941,159.268
C00620=1037.471,416.628,-140.841,174.531,45.947,159.271
C00621=1037.482,416.874,-140.889,174.544,45.953,159.274
C00622=1037.493,417.119,-140.935,174.555,45.959,159.277
C00623=1037.504,417.364,-140.984,174.566,45.965,159.280
C00624=1037.514,417.609,-141.031,174.578,45.971,159.283
C00625=1037.525,417.855,-141.078,174.589,45.978,159.286
C00626=1037.536,418.100,-141.126,174.601,45.983,159.289
C00627=1037.547,418.344,-141.174,174.613,45.990,159.292
C00628=1037.558,418.590,-141.221,174.625,45.996,159.295
C00629=1037.568,418.835,-141.269,174.636,46.002,159.298
C00630=1037.579,419.080,-141.317,174.647,46.009,159.301
C00631=1037.590,419.326,-141.365,174.659,46.015,159.304
C00632=1037.601,419.571,-141.413,174.671,46.021,159.307
C00633=1037.611,419.816,-141.461,174.683,46.027,159.310
C00634=1037.622,420.061,-141.509,174.695,46.034,159.313
C00635=1037.633,420.306,-141.557,174.706,46.040,159.316
C00636=1037.644,420.551,-141.605,174.719,46.046,159.320
C00637=1037.655,420.796,-141.654,174.731,46.052,159.323
C00638=1037.666,421.042,-141.702,174.742,46.059,159.326
C00639=1037.677,421.278,-141.748,174.755,46.065,159.329
C00640=1037.688,421.514,-141.794,174.766,46.071,159.332
C00641=1037.697,421.750,-141.841,174.778,46.078,159.335
C00642=1037.709,421.986,-141.887,174.789,46.084,159.338
C00643=1037.720,422.223,-141.934,174.802,46.090,159.341
C00644=1037.730,422.459,-141.981,174.813,46.097,159.344
C00645=1037.741,422.695,-142.027,174.825,46.102,159.347
C00646=1037.752,422.932,-142.075,174.837,46.109,159.350
C00647=1037.763,423.177,-142.123,174.849,46.116,159.354
C00648=1037.775,423.421,-142.171,174.862,46.122,159.357
C00649=1037.786,423.667,-142.220,174.875,46.129,159.360
C00650=1037.797,423.912,-142.269,174.887,46.135,159.363
C00651=1037.808,424.157,-142.317,174.900,46.142,159.367
C00652=1037.819,424.402,-142.366,174.912,46.149,159.370
C00653=1037.831,424.647,-142.416,174.925,46.155,159.373
C00654=1037.842,424.891,-142.465,174.938,46.162,159.377
C00655=1037.853,425.136,-142.514,174.950,46.169,159.380
C00656=1037.865,425.381,-142.563,174.963,46.176,159.384
C00657=1037.875,425.627,-142.611,174.976,46.182,159.387
C00658=1037.887,425.871,-142.661,174.988,46.189,159.390
C00659=1037.898,426.115,-142.710,175.001,46.196,159.394
C00660=1037.910,426.361,-142.760,175.014,46.203,159.397
C00661=1037.922,426.606,-142.809,175.027,46.210,159.401
C00662=1037.933,426.850,-142.858,175.041,46.217,159.404
C00663=1037.944,427.095,-142.907,175.054,46.224,159.408
C00664=1037.956,427.340,-142.957,175.066,46.231,159.411
C00665=1037.967,427.585,-143.006,175.080,46.238,159.415
C00666=1037.979,427.830,-143.055,175.093,46.244,159.418
C00667=1037.991,428.074,-143.105,175.106,46.252,159.422
C00668=1038.002,428.320,-143.155,175.119,46.259,159.425
C00669=1038.014,428.564,-143.205,175.133,46.266,159.429
C00670=1038.025,428.809,-143.255,175.146,46.273,159.432
C00671=1038.037,429.054,-143.304,175.159,46.280,159.436
C00672=1038.049,429.298,-143.355,175.173,46.287,159.439
C00673=1038.060,429.543,-143.405,175.186,46.294,159.443
C00674=1038.072,429.788,-143.455,175.200,46.301,159.447
C00675=1038.083,430.032,-143.505,175.214,46.309,159.450
C00676=1038.095,430.277,-143.555,175.228,46.316,159.454
C00677=1038.107,430.522,-143.606,175.241,46.323,159.458
C00678=1038.119,430.766,-143.656,175.255,46.330,159.461
C00679=1038.131,431.011,-143.706,175.268,46.338,159.465
C00680=1038.143,431.256,-143.757,175.283,46.345,159.469
C00681=1038.154,431.500,-143.806,175.297,46.353,159.473
C00682=1038.166,431.745,-143.858,175.310,46.360,159.476
C00683=1038.179,431.990,-143.908,175.324,46.367,159.480
C00684=1038.191,432.234,-143.958,175.339,46.375,159.484
C00685=1038.202,432.478,-144.009,175.353,46.382,159.488
C00686=1038.214,432.723,-144.059,175.366,46.390,159.491
C00687=1038.226,432.967,-144.110,175.381,46.397,159.495
C00688=1038.239,433.212,-144.161,175.395,46.404,159.499
C00689=1038.250,433.457,-144.212,175.410,46.412,159.503
C00690=1038.263,433.701,-144.263,175.424,46.419,159.507
C00691=1038.275,433.946,-144.313,175.439,46.427,159.511
C00692=1038.287,434.190,-144.364,175.453,46.435,159.515
C00693=1038.300,434.435,-144.415,175.468,46.442,159.519
C00694=1038.312,434.679,-144.466,175.482,46.450,159.523
C00695=1038.324,434.923,-144.517,175.497,46.458,159.526
C00696=1038.336,435.168,-144.569,175.512,46.466,159.530
C00697=1038.349,435.412,-144.620,175.526,46.473,159.534
C00698=1038.361,435.657,-144.671,175.541,46.481,159.538
C00699=1038.373,435.897,-144.721,175.555,46.489,159.542
C00700=1038.385,436.137,-144.773,175.570,46.496,159.546
C00701=1038.398,436.377,-144.823,175.585,46.504,159.550
C00702=1038.409,436.617,-144.873,175.599,46.512,159.554
C00703=1038.422,436.857,-144.924,175.614,46.519,159.558
C00704=1038.435,437.097,-144.975,175.630,46.527,159.562
C00705=1038.447,437.337,-145.026,175.644,46.535,159.567
C00706=1038.459,437.576,-145.077,175.659,46.543,159.571
C00707=1038.471,437.821,-145.129,175.674,46.551,159.575
C00708=1038.484,438.065,-145.181,175.690,46.559,159.579
C00709=1038.497,438.310,-145.233,175.705,46.567,159.583
C00710=1038.509,438.553,-145.285,175.721,46.575,159.587
C00711=1038.522,438.798,-145.337,175.736,46.583,159.591
C00712=1038.534,439.042,-145.389,175.752,46.591,159.596
C00713=1038.548,439.286,-145.441,175.767,46.599,159.600
C00714=1038.560,439.530,-145.493,175.783,46.607,159.604
C00715=1038.573,439.775,-145.546,175.798,46.616,159.609
C00716=1038.586,440.019,-145.598,175.814,46.624,159.613
C00717=1038.599,440.263,-145.650,175.830,46.632,159.617
C00718=1038.612,440.507,-145.703,175.847,46.640,159.622
C00719=1038.624,440.751,-145.756,175.862,46.648,159.626
C00720=1038.638,440.995,-145.809,175.878,46.657,159.631
C00721=1038.650,441.239,-145.861,175.894,46.665,159.635
C00722=1038.663,441.483,-145.914,175.911,46.673,159.639
C00723=1038.676,441.727,-145.967,175.927,46.682,159.644
C00724=1038.689,441.972,-146.020,175.943,46.690,159.648
C00725=1038.703,442.215,-146.072,175.960,46.699,159.653
C00726=1038.716,442.459,-146.126,175.976,46.707,159.657
C00727=1038.729,442.703,-146.179,175.993,46.716,159.662
C00728=1038.742,442.947,-146.232,176.009,46.724,159.666
C00729=1038.755,443.191,-146.285,176.026,46.733,159.671
C00730=1038.768,443.435,-146.338,176.042,46.741,159.676
C00731=1038.781,443.679,-146.392,176.059,46.750,159.680
C00732=1038.795,443.923,-146.444,176.076,46.759,159.685
C00733=1038.808,444.166,-146.498,176.092,46.767,159.689
C00734=1038.821,444.410,-146.551,176.110,46.776,159.694
C00735=1038.835,444.653,-146.604,176.126,46.784,159.699
C00736=1038.850,444.896,-146.656,176.144,46.793,159.703
C00737=1038.865,445.140,-146.709,176.160,46.801,159.708
C00738=1038.880,445.384,-146.761,176.178,46.810,159.713
C00739=1038.896,445.627,-146.812,176.196,46.818,159.717
C00740=1038.912,445.871,-146.862,176.212,46.826,159.722
C00741=1038.929,446.114,-146.912,176.229,46.834,159.726
C00742=1038.947,446.359,-146.962,176.248,46.842,159.731
C00743=1038.966,446.602,-147.011,176.265,46.850,159.736
C00744=1038.984,446.846,-147.061,176.283,46.857,159.740
C00745=1039.004,447.091,-147.109,176.301,46.865,159.745
C00746=1039.024,447.335,-147.157,176.318,46.872,159.749
C00747=1039.045,447.580,-147.204,176.336,46.880,159.754
C00748=1039.066,447.824,-147.252,176.355,46.887,159.758
C00749=1039.087,448.068,-147.299,176.372,46.894,159.762
C00750=1039.109,448.313,-147.344,176.390,46.901,159.767
C00751=1039.132,448.558,-147.390,176.409,46.908,159.771
C00752=1039.156,448.803,-147.436,176.427,46.915,159.776
C00753=1039.180,449.048,-147.480,176.445,46.923,159.780
C00754=1039.204,449.292,-147.525,176.464,46.929,159.785
C00755=1039.229,449.538,-147.569,176.482,46.936,159.789
C00756=1039.255,449.782,-147.612,176.501,46.942,159.793
C00757=1039.280,450.028,-147.655,176.520,46.949,159.798
C00758=1039.307,450.273,-147.698,176.539,46.955,159.802
C00759=1039.354,450.687,-147.768,176.571,46.966,159.809
C00760=1039.402,451.102,-147.838,176.603,46.976,159.817
C00761=1039.452,451.515,-147.906,176.635,46.986,159.824
C00762=1039.502,451.927,-147.972,176.668,46.996,159.831
C00763=1039.208,451.977,-148.292,176.671,47.071,159.854
C00764=1039.158,451.579,-148.228,176.640,47.061,159.847
C00765=1039.110,451.180,-148.163,176.608,47.052,159.840
C00766=1039.064,450.780,-148.096,176.577,47.042,159.833
C00767=1039.019,450.380,-148.028,176.546,47.032,159.826
C00768=1038.991,450.136,-147.986,176.527,47.025,159.822
C00769=1038.965,449.890,-147.943,176.508,47.019,159.817
C00770=1038.939,449.645,-147.900,176.489,47.012,159.813
C00771=1038.913,449.400,-147.857,176.470,47.006,159.809
C00772=1038.889,449.155,-147.813,176.452,46.999,159.804
C00773=1038.864,448.910,-147.768,176.433,46.993,159.800
C00774=1038.841,448.665,-147.723,176.415,46.986,159.795
C00775=1038.818,448.421,-147.677,176.397,46.979,159.791
C00776=1038.795,448.175,-147.631,176.378,46.972,159.786
C00777=1038.773,447.931,-147.585,176.359,46.965,159.782
C00778=1038.752,447.686,-147.538,176.342,46.957,159.778
C00779=1038.731,447.442,-147.491,176.324,46.950,159.773
C00780=1038.710,447.197,-147.443,176.306,46.943,159.769
C00781=1038.691,446.953,-147.394,176.289,46.935,159.764
C00782=1038.671,446.709,-147.347,176.270,46.928,159.760
C00783=1038.653,446.465,-147.297,176.253,46.920,159.755
C00784=1038.634,446.221,-147.247,176.235,46.912,159.750
C00785=1038.617,445.977,-147.197,176.217,46.905,159.746
C00786=1038.600,445.734,-147.147,176.200,46.897,159.741
C00787=1038.584,445.490,-147.096,176.183,46.888,159.737
C00788=1038.568,445.246,-147.044,176.165,46.880,159.732
C00789=1038.553,445.002,-146.993,176.148,46.872,159.728
C00790=1038.539,444.760,-146.940,176.131,46.864,159.723
C00791=1038.524,444.516,-146.888,176.114,46.856,159.718
C00792=1038.511,444.273,-146.835,176.097,46.847,159.714
C00793=1038.497,444.029,-146.781,176.080,46.838,159.709
C00794=1038.483,443.786,-146.728,176.063,46.830,159.704
C00795=1038.471,443.543,-146.675,176.046,46.821,159.700
C00796=1038.457,443.298,-146.622,176.030,46.813,159.695
C00797=1038.444,443.054,-146.568,176.013,46.804,159.691
C00798=1038.431,442.810,-146.515,175.996,46.796,159.686
C00799=1038.417,442.567,-146.463,175.979,46.788,159.681
C00800=1038.404,442.323,-146.409,175.963,46.779,159.677
C00801=1038.391,442.079,-146.356,175.946,46.771,159.672
C00802=1038.378,441.835,-146.303,175.930,46.763,159.668
C00803=1038.366,441.591,-146.251,175.914,46.754,159.663
C00804=1038.353,441.347,-146.198,175.897,46.746,159.659
C00805=1038.339,441.103,-146.145,175.882,46.737,159.655
C00806=1038.326,440.859,-146.093,175.866,46.729,159.650
C00807=1038.313,440.615,-146.039,175.849,46.721,159.646
C00808=1038.301,440.371,-145.987,175.833,46.713,159.641
C00809=1038.288,440.127,-145.934,175.817,46.705,159.637
C00810=1038.275,439.882,-145.882,175.802,46.696,159.633
C00811=1038.261,439.638,-145.830,175.786,46.688,159.628
C00812=1038.249,439.394,-145.778,175.770,46.680,159.624
C00813=1038.236,439.149,-145.725,175.755,46.672,159.620
C00814=1038.224,438.906,-145.673,175.739,46.664,159.615
C00815=1038.211,438.661,-145.621,175.722,46.656,159.611
C00816=1038.198,438.417,-145.569,175.708,46.648,159.607
C00817=1038.186,438.173,-145.516,175.692,46.640,159.603
C00818=1038.173,437.929,-145.465,175.677,46.632,159.599
C00819=1038.160,437.685,-145.412,175.661,46.625,159.594
C00820=1038.148,437.444,-145.362,175.646,46.617,159.590
C00821=1038.136,437.203,-145.310,175.631,46.609,159.586
C00822=1038.123,436.963,-145.259,175.616,46.601,159.582
C00823=1038.111,436.722,-145.209,175.601,46.593,159.578
C00824=1038.098,436.481,-145.158,175.586,46.586,159.574
C00825=1038.086,436.241,-145.107,175.571,46.578,159.570
C00826=1038.075,436.000,-145.056,175.557,46.571,159.566
C00827=1038.062,435.759,-145.005,175.542,46.563,159.562
C00828=1038.049,435.514,-144.954,175.527,46.555,159.558
C00829=1038.037,435.270,-144.903,175.513,46.548,159.554
C00830=1038.025,435.025,-144.851,175.498,46.540,159.550
C00831=1038.013,434.781,-144.801,175.483,46.532,159.546
C00832=1038.001,434.537,-144.749,175.468,46.524,159.542
C00833=1037.988,434.292,-144.698,175.453,46.517,159.538
C00834=1037.976,434.048,-144.648,175.439,46.510,159.534
C00835=1037.964,433.804,-144.596,175.424,46.502,159.530
C00836=1037.951,433.559,-144.546,175.410,46.495,159.527
C00837=1037.940,433.314,-144.495,175.395,46.487,159.523
C00838=1037.927,433.070,-144.444,175.381,46.480,159.519
C00839=1037.915,432.825,-144.394,175.368,46.472,159.515
C00840=1037.903,432.581,-144.342,175.353,46.465,159.511
C00841=1037.890,432.336,-144.292,175.339,46.458,159.508
C00842=1037.879,432.091,-144.241,175.325,46.450,159.504
C00843=1037.866,431.847,-144.191,175.310,46.443,159.500
C00844=1037.855,431.603,-144.141,175.297,46.436,159.496
C00845=1037.843,431.358,-144.090,175.283,46.428,159.492
C00846=1037.830,431.113,-144.040,175.268,46.421,159.489
C00847=1037.819,430.868,-143.989,175.254,46.414,159.485
C00848=1037.807,430.624,-143.939,175.241,46.406,159.481
C00849=1037.795,430.379,-143.889,175.227,46.400,159.478
C00850=1037.784,430.135,-143.839,175.214,46.392,159.474
C00851=1037.772,429.890,-143.789,175.200,46.385,159.470
C00852=1037.760,429.645,-143.738,175.186,46.378,159.467
C00853=1037.748,429.401,-143.688,175.172,46.371,159.463
C00854=1037.736,429.156,-143.638,175.159,46.364,159.459
C00855=1037.725,428.911,-143.588,175.145,46.357,159.456
C00856=1037.714,428.667,-143.539,175.132,46.350,159.452
C00857=1037.702,428.421,-143.488,175.118,46.343,159.448
C00858=1037.690,428.177,-143.438,175.105,46.336,159.445
C00859=1037.678,427.932,-143.389,175.092,46.329,159.441
C00860=1037.667,427.687,-143.339,175.078,46.322,159.438
C00861=1037.655,427.442,-143.289,175.065,46.315,159.434
C00862=1037.644,427.197,-143.240,175.052,46.308,159.431
C00863=1037.632,426.953,-143.191,175.038,46.301,159.427
C00864=1037.621,426.707,-143.141,175.026,46.294,159.424
C00865=1037.609,426.463,-143.092,175.013,46.287,159.421
C00866=1037.598,426.218,-143.043,175.000,46.281,159.417
C00867=1037.587,425.973,-142.993,174.986,46.274,159.414
C00868=1037.575,425.728,-142.944,174.974,46.267,159.410
C00869=1037.563,425.483,-142.895,174.961,46.261,159.407
C00870=1037.552,425.238,-142.846,174.948,46.254,159.404
C00871=1037.541,424.993,-142.796,174.935,46.247,159.400
C00872=1037.530,424.748,-142.747,174.923,46.240,159.397
C00873=1037.518,424.504,-142.698,174.910,46.233,159.393
C00874=1037.507,424.258,-142.650,174.897,46.227,159.390
C00875=1037.496,424.014,-142.601,174.885,46.220,159.387
C00876=1037.484,423.769,-142.552,174.872,46.213,159.383
C00877=1037.473,423.524,-142.504,174.859,46.207,159.380
C00878=1037.462,423.279,-142.455,174.847,46.201,159.377
C00879=1037.451,423.033,-142.407,174.834,46.194,159.374
C00880=1037.440,422.796,-142.359,174.822,46.188,159.371
C00881=1037.430,422.559,-142.313,174.811,46.182,159.368
C00882=1037.419,422.321,-142.265,174.798,46.176,159.364
C00883=1037.407,422.085,-142.219,174.787,46.169,159.361
C00884=1037.397,421.847,-142.172,174.775,46.163,159.358
C00885=1037.386,421.610,-142.125,174.763,46.157,159.355
C00886=1037.375,421.372,-142.078,174.751,46.151,159.352
C00887=1037.365,421.135,-142.031,174.740,46.144,159.349
C00888=1037.354,420.890,-141.983,174.727,46.138,159.346
C00889=1037.342,420.645,-141.935,174.715,46.132,159.343
C00890=1037.331,420.400,-141.887,174.703,46.126,159.340
C00891=1037.320,420.155,-141.839,174.691,46.119,159.336
C00892=1037.309,419.910,-141.791,174.679,46.113,159.333
C00893=1037.299,419.665,-141.743,174.668,46.107,159.330
C00894=1037.288,419.419,-141.695,174.655,46.101,159.327
C00895=1037.277,419.174,-141.647,174.643,46.094,159.324
C00896=1037.266,418.929,-141.599,174.632,46.088,159.321
C00897=1037.255,418.684,-141.551,174.620,46.082,159.318
C00898=1037.245,418.438,-141.503,174.608,46.076,159.315
C00899=1037.233,418.193,-141.456,174.596,46.070,159.312
C00900=1037.223,417.948,-141.408,174.585,46.064,159.309
C00901=1037.213,417.703,-141.361,174.573,46.058,159.306
C00902=1037.202,417.457,-141.313,174.562,46.051,159.303
C00903=1037.191,417.213,-141.265,174.550,46.046,159.300
C00904=1037.180,416.967,-141.218,174.539,46.040,159.297
C00905=1037.170,416.722,-141.171,174.528,46.033,159.294
C00906=1037.159,416.476,-141.124,174.515,46.028,159.291
C00907=1037.148,416.231,-141.077,174.504,46.022,159.288
C00908=1037.137,415.986,-141.029,174.494,46.016,159.286
C00909=1037.126,415.741,-140.982,174.482,46.010,159.283
C00910=1037.116,415.495,-140.934,174.470,46.004,159.280
C00911=1037.105,415.250,-140.887,174.459,45.998,159.277
C00912=1037.094,415.005,-140.841,174.448,45.993,159.274
C00913=1037.084,414.760,-140.793,174.437,45.987,159.271
C00914=1037.074,414.514,-140.747,174.426,45.981,159.268
C00915=1037.063,414.268,-140.700,174.415,45.975,159.265
C00916=1037.053,414.023,-140.653,174.404,45.969,159.263
C00917=1037.042,413.778,-140.606,174.392,45.963,159.260
C00918=1037.032,413.532,-140.559,174.381,45.958,159.257
C00919=1037.022,413.287,-140.512,174.370,45.952,159.254
C00920=1037.011,413.042,-140.466,174.359,45.946,159.251
C00921=1037.001,412.796,-140.419,174.349,45.940,159.249
C00922=1036.990,412.551,-140.373,174.338,45.935,159.246
C00923=1036.980,412.305,-140.325,174.327,45.929,159.243
C00924=1036.970,412.060,-140.279,174.316,45.924,159.240
C00925=1036.959,411.815,-140.232,174.305,45.918,159.238
C00926=1036.949,411.569,-140.186,174.295,45.913,159.235
C00927=1036.939,411.324,-140.140,174.284,45.907,159.232
C00928=1036.929,411.078,-140.094,174.273,45.901,159.230
C00929=1036.918,410.833,-140.047,174.262,45.896,159.227
C00930=1036.908,410.587,-140.001,174.252,45.890,159.224
C00931=1036.898,410.341,-139.955,174.241,45.885,159.222
C00932=1036.887,410.096,-139.909,174.231,45.879,159.219
C00933=1036.876,409.850,-139.863,174.220,45.874,159.216
C00934=1036.866,409.605,-139.817,174.209,45.869,159.214
C00935=1036.857,409.359,-139.771,174.199,45.863,159.211
C00936=1036.846,409.114,-139.725,174.188,45.858,159.208
C00937=1036.835,408.868,-139.679,174.179,45.853,159.206
C00938=1036.825,408.623,-139.634,174.168,45.847,159.203
C00939=1036.816,408.377,-139.588,174.158,45.842,159.201
C00940=1036.806,408.144,-139.545,174.148,45.837,159.198
C00941=1036.796,407.911,-139.501,174.138,45.832,159.196
C00942=1036.787,407.679,-139.457,174.128,45.827,159.193
C00943=1036.777,407.445,-139.414,174.118,45.822,159.191
C00944=1036.768,407.212,-139.371,174.109,45.817,159.189
C00945=1036.758,406.979,-139.328,174.099,45.812,159.186
C00946=1036.749,406.746,-139.285,174.089,45.807,159.184
C00947=1036.739,406.513,-139.241,174.080,45.802,159.181
C00948=1036.729,406.267,-139.196,174.069,45.797,159.179
C00949=1036.719,406.022,-139.151,174.060,45.791,159.176
C00950=1036.709,405.776,-139.105,174.050,45.787,159.174
C00951=1036.699,405.531,-139.059,174.039,45.782,159.171
C00952=1036.689,405.285,-139.014,174.030,45.776,159.169
C00953=1036.679,405.039,-138.969,174.020,45.771,159.166
C00954=1036.670,404.794,-138.923,174.010,45.766,159.164
C00955=1036.660,404.548,-138.878,174.000,45.761,159.161
C00956=1036.650,404.302,-138.833,173.990,45.756,159.159
C00957=1036.640,404.057,-138.788,173.980,45.751,159.157
C00958=1036.631,403.811,-138.743,173.970,45.746,159.154
C00959=1036.621,403.565,-138.697,173.961,45.741,159.152
C00960=1036.611,403.320,-138.652,173.950,45.736,159.149
C00961=1036.601,403.074,-138.607,173.941,45.731,159.147
C00962=1036.592,402.829,-138.563,173.932,45.726,159.145
C00963=1036.582,402.583,-138.518,173.922,45.721,159.142
C00964=1036.572,402.336,-138.473,173.912,45.716,159.140
C00965=1036.563,402.091,-138.428,173.902,45.711,159.138
C00966=1036.553,401.845,-138.383,173.893,45.706,159.135
C00967=1036.544,401.600,-138.338,173.883,45.701,159.133
C00968=1036.534,401.353,-138.294,173.874,45.697,159.131
C00969=1036.524,401.108,-138.249,173.865,45.692,159.128
C00970=1036.515,400.862,-138.204,173.854,45.687,159.126
C00971=1036.505,400.616,-138.160,173.845,45.682,159.124
C00972=1036.496,400.371,-138.115,173.836,45.677,159.122
C00973=1036.485,400.125,-138.072,173.826,45.673,159.119
C00974=1036.476,399.879,-138.027,173.817,45.668,159.117
C00975=1036.466,399.633,-137.983,173.808,45.663,159.115
C00976=1036.457,399.388,-137.938,173.798,45.658,159.112
C00977=1036.447,399.142,-137.894,173.789,45.654,159.110
C00978=1036.438,398.895,-137.850,173.780,45.649,159.108
C00979=1036.428,398.650,-137.805,173.771,45.644,159.106
C00980=1036.418,398.404,-137.762,173.761,45.640,159.103
C00981=1036.408,398.158,-137.718,173.752,45.635,159.101
C00982=1036.400,397.913,-137.674,173.743,45.631,159.099
C00983=1036.390,397.666,-137.630,173.734,45.626,159.097
C00984=1036.381,397.420,-137.586,173.724,45.621,159.095
C00985=1036.370,397.175,-137.541,173.715,45.617,159.092
C00986=1036.362,396.930,-137.498,173.706,45.612,159.090
C00987=1036.352,396.684,-137.454,173.697,45.608,159.088
C00988=1036.343,396.437,-137.409,173.688,45.603,159.086
C00989=1036.333,396.192,-137.366,173.679,45.598,159.084
C00990=1036.324,395.946,-137.323,173.670,45.594,159.082
C00991=1036.315,395.699,-137.279,173.661,45.590,159.080
C00992=1036.305,395.453,-137.235,173.651,45.585,159.077
C00993=1036.297,395.208,-137.191,173.642,45.581,159.075
C00994=1036.286,394.962,-137.147,173.634,45.577,159.073
C00995=1036.278,394.717,-137.104,173.625,45.572,159.071
C00996=1036.268,394.470,-137.060,173.616,45.568,159.069
C00997=1036.258,394.224,-137.017,173.607,45.563,159.067
C00998=1036.250,393.978,-136.974,173.598,45.559,159.065
C00999=1036.240,393.732,-136.930,173.589,45.554,159.063
C01000=1036.232,393.509,-136.891,173.582,45.550,159.061
C01001=1036.224,393.286,-136.851,173.573,45.547,159.059
C01002=1036.215,393.063,-136.813,173.566,45.543,159.057
C01003=1036.207,392.840,-136.773,173.557,45.539,159.055
C01004=1036.198,392.618,-136.734,173.550,45.535,159.054
C01005=1036.190,392.395,-136.694,173.542,45.531,159.052
C01006=1036.182,392.172,-136.656,173.534,45.528,159.050
C01007=1036.174,391.949,-136.616,173.526,45.524,159.048
C01008=1036.164,391.703,-136.574,173.518,45.519,159.046
C01009=1036.155,391.456,-136.530,173.509,45.515,159.044
C01010=1036.146,391.211,-136.487,173.500,45.511,159.042
C01011=1036.137,390.965,-136.444,173.492,45.507,159.040
C01012=1036.127,390.719,-136.401,173.484,45.503,159.038
C01013=1036.119,390.473,-136.358,173.475,45.498,159.036
C01014=1036.110,390.227,-136.316,173.467,45.494,159.034
C01015=1036.100,389.980,-136.273,173.458,45.490,159.032
C01016=1036.091,389.734,-136.230,173.449,45.486,159.030
C01017=1036.083,389.488,-136.187,173.441,45.482,159.028
C01018=1036.073,389.242,-136.144,173.433,45.478,159.026
C01019=1036.064,388.996,-136.102,173.424,45.474,159.024
C01020=1036.055,388.750,-136.059,173.416,45.470,159.022
C01021=1036.046,388.504,-136.016,173.407,45.466,159.020
C01022=1036.037,388.257,-135.974,173.399,45.462,159.018
C01023=1036.028,388.011,-135.931,173.391,45.458,159.017
C01024=1036.019,387.766,-135.889,173.383,45.454,159.015
C01025=1036.010,387.519,-135.846,173.374,45.450,159.013
C01026=1036.001,387.273,-135.804,173.366,45.446,159.011
C01027=1035.992,387.027,-135.762,173.358,45.442,159.009
C01028=1035.982,386.780,-135.720,173.350,45.438,159.007
C01029=1035.974,386.534,-135.677,173.341,45.434,159.005
C01030=1035.965,386.288,-135.635,173.334,45.430,159.004
C01031=1035.956,386.042,-135.592,173.325,45.427,159.002
C01032=1035.947,385.796,-135.551,173.317,45.423,159.000
C01033=1035.938,385.550,-135.508,173.309,45.419,158.998
C01034=1035.929,385.304,-135.467,173.301,45.415,158.996
C01035=1035.920,385.057,-135.425,173.292,45.411,158.994
C01036=1035.911,384.811,-135.382,173.285,45.408,158.993
C01037=1035.902,384.565,-135.340,173.277,45.404,158.991
C01038=1035.893,384.319,-135.298,173.268,45.400,158.989
C01039=1035.884,384.072,-135.257,173.261,45.396,158.987
C01040=1035.875,383.826,-135.215,173.252,45.393,158.985
C01041=1035.866,383.580,-135.172,173.245,45.389,158.983
C01042=1035.857,383.334,-135.131,173.237,45.385,158.982
C01043=1035.848,383.087,-135.089,173.229,45.381,158.980
C01044=1035.840,382.841,-135.047,173.221,45.377,158.978
C01045=1035.831,382.594,-135.005,173.214,45.374,158.976
C01046=1035.823,382.349,-134.964,173.205,45.370,158.975
C01047=1035.814,382.102,-134.922,173.198,45.367,158.973
C01048=1035.804,381.821,-134.874,173.188,45.362,158.971
C01049=1035.794,381.540,-134.827,173.180,45.358,158.969
C01050=1035.784,381.258,-134.779,173.171,45.354,158.967
C01051=1035.775,380.977,-134.732,173.162,45.350,158.965
C01052=1035.766,380.731,-134.690,173.154,45.346,158.963
C01053=1035.757,380.484,-134.649,173.147,45.343,158.962
C01054=1035.748,380.239,-134.607,173.139,45.340,158.960
C01055=1035.739,379.992,-134.566,173.131,45.335,158.958
C01056=1035.731,379.745,-134.525,173.123,45.332,158.956
C01057=1035.723,379.499,-134.483,173.116,45.329,158.955
C01058=1035.714,379.253,-134.441,173.108,45.325,158.953
C01059=1035.706,379.006,-134.400,173.100,45.322,158.951
C01060=1035.693,378.631,-134.338,173.089,45.316,158.949
C01061=1035.680,378.254,-134.274,173.077,45.311,158.946
C01062=1035.667,377.877,-134.211,173.066,45.306,158.944
C01063=1035.654,377.502,-134.149,173.055,45.301,158.941
C01064=1035.645,377.255,-134.108,173.047,45.297,158.940
C01065=1035.636,377.008,-134.067,173.039,45.294,158.938
C01066=1035.627,376.763,-134.026,173.032,45.290,158.936
C01067=1035.619,376.516,-133.985,173.024,45.287,158.935
C01068=1035.611,376.269,-133.944,173.017,45.283,158.933
C01069=1035.601,376.023,-133.904,173.010,45.280,158.932
C01070=1035.593,375.776,-133.863,173.002,45.277,158.930
C01071=1035.584,375.530,-133.821,172.995,45.274,158.928
C01072=1035.576,375.284,-133.781,172.988,45.271,158.927
C01073=1035.568,375.037,-133.740,172.981,45.267,158.925
C01074=1035.559,374.791,-133.700,172.972,45.264,158.923
C01075=1035.551,374.544,-133.659,172.965,45.261,158.922
C01076=1035.542,374.297,-133.618,172.958,45.257,158.920
C01077=1035.534,374.051,-133.577,172.951,45.254,158.919
C01078=1035.525,373.805,-133.537,172.943,45.251,158.917
C01079=1035.517,373.558,-133.496,172.936,45.248,158.916
C01080=1035.509,373.311,-133.457,172.929,45.244,158.914
C01081=1035.500,373.064,-133.415,172.922,45.241,158.913
C01082=1035.492,372.818,-133.375,172.915,45.238,158.911
C01083=1035.484,372.572,-133.335,172.908,45.235,158.910
C01084=1035.475,372.325,-133.294,172.900,45.232,158.908
C01085=1035.467,372.078,-133.254,172.893,45.229,158.907
C01086=1035.459,371.832,-133.214,172.886,45.226,158.905
C01087=1035.450,371.586,-133.173,172.879,45.222,158.903
C01088=1035.442,371.339,-133.132,172.872,45.219,158.902
C01089=1035.434,371.092,-133.092,172.865,45.216,158.901
C01090=1035.425,370.846,-133.052,172.858,45.213,158.899
C01091=1035.418,370.599,-133.012,172.851,45.210,158.897
C01092=1035.410,370.353,-132.972,172.844,45.207,158.896
C01093=1035.401,370.106,-132.932,172.836,45.204,158.894
C01094=1035.393,369.859,-132.891,172.829,45.201,158.893
C01095=1035.385,369.612,-132.851,172.822,45.198,158.892
C01096=1035.376,369.366,-132.811,172.816,45.195,158.890
C01097=1035.368,369.120,-132.772,172.809,45.192,158.889
C01098=1035.359,368.872,-132.732,172.802,45.189,158.887
C01099=1035.351,368.626,-132.692,172.795,45.186,158.886
C01100=1035.343,368.379,-132.652,172.788,45.183,158.884
C01101=1035.334,368.133,-132.613,172.781,45.180,158.883
C01102=1035.327,367.886,-132.573,172.774,45.177,158.881
C01103=1035.318,367.639,-132.533,172.767,45.174,158.880
C01104=1035.309,367.393,-132.493,172.760,45.171,158.879
C01105=1035.302,367.146,-132.453,172.753,45.168,158.877
C01106=1035.293,366.900,-132.414,172.747,45.166,158.876
C01107=1035.285,366.653,-132.374,172.740,45.163,158.874
C01108=1035.277,366.406,-132.335,172.733,45.160,158.873
C01109=1035.269,366.160,-132.295,172.726,45.157,158.871
C01110=1035.261,365.913,-132.256,172.720,45.154,158.870
C01111=1035.252,365.666,-132.216,172.713,45.151,158.869
C01112=1035.245,365.419,-132.176,172.706,45.148,158.867
C01113=1035.236,365.173,-132.137,172.699,45.146,158.866
C01114=1035.228,364.926,-132.098,172.692,45.143,158.865
C01115=1035.220,364.679,-132.058,172.685,45.140,158.863
C01116=1035.207,364.288,-131.995,172.676,45.135,158.861
C01117=1035.195,363.898,-131.933,172.665,45.131,158.859
C01118=1035.182,363.508,-131.871,172.654,45.127,158.857
C01119=1035.169,363.116,-131.809,172.643,45.123,158.855
C01120=1035.161,362.870,-131.770,172.638,45.120,158.853
C01121=1035.153,362.624,-131.731,172.631,45.117,158.852
C01122=1035.146,362.376,-131.691,172.624,45.114,158.851
C01123=1035.137,362.130,-131.652,172.617,45.111,158.849
C01124=1035.129,361.883,-131.613,172.611,45.109,158.848
C01125=1035.121,361.636,-131.573,172.604,45.106,158.847
C01126=1035.113,361.390,-131.535,172.598,45.103,158.845
C01127=1035.105,361.143,-131.496,172.592,45.101,158.844
C01128=1035.097,360.895,-131.457,172.585,45.098,158.843
C01129=1035.089,360.649,-131.418,172.578,45.096,158.842
C01130=1035.082,360.402,-131.379,172.571,45.093,158.840
C01131=1035.073,360.155,-131.340,172.566,45.090,158.839
C01132=1035.065,359.908,-131.301,172.559,45.088,158.838
C01133=1035.058,359.662,-131.263,172.553,45.085,158.836
C01134=1035.049,359.415,-131.224,172.546,45.083,158.835
C01135=1035.041,359.168,-131.185,172.540,45.080,158.834
C01136=1035.033,358.921,-131.146,172.534,45.078,158.833
C01137=1035.025,358.674,-131.108,172.527,45.076,158.831
C01138=1035.017,358.427,-131.070,172.520,45.073,158.830
C01139=1035.009,358.181,-131.031,172.515,45.070,158.829
C01140=1035.001,357.934,-130.992,172.508,45.068,158.828
C01141=1034.993,357.686,-130.953,172.502,45.066,158.826
C01142=1034.986,357.440,-130.915,172.495,45.063,158.825
C01143=1034.978,357.192,-130.876,172.489,45.060,158.824
C01144=1034.971,356.946,-130.838,172.483,45.058,158.823
C01145=1034.962,356.699,-130.799,172.476,45.056,158.821
C01146=1034.954,356.451,-130.761,172.471,45.053,158.820
C01147=1034.947,356.205,-130.722,172.464,45.050,158.819
C01148=1034.939,355.958,-130.684,172.457,45.048,158.818
C01149=1034.931,355.711,-130.645,172.452,45.046,158.817
C01150=1034.923,355.464,-130.607,172.445,45.043,158.815
C01151=1034.915,355.217,-130.570,172.439,45.041,158.814
C01152=1034.907,354.970,-130.531,172.434,45.039,158.813
C01153=1034.899,354.723,-130.493,172.427,45.036,158.812
C01154=1034.891,354.476,-130.454,172.420,45.034,158.810
C01155=1034.884,354.229,-130.417,172.415,45.032,158.809
C01156=1034.876,353.982,-130.378,172.408,45.029,158.808
C01157=1034.867,353.736,-130.341,172.402,45.027,158.807
C01158=1034.860,353.489,-130.302,172.396,45.025,158.806
C01159=1034.852,353.241,-130.264,172.390,45.022,158.805
C01160=1034.844,352.995,-130.226,172.384,45.020,158.804
C01161=1034.837,352.747,-130.188,172.378,45.018,158.802
C01162=1034.829,352.500,-130.150,172.372,45.016,158.801
C01163=1034.821,352.254,-130.113,172.366,45.013,158.800
C01164=1034.813,352.006,-130.075,172.360,45.011,158.799
C01165=1034.805,351.760,-130.036,172.354,45.009,158.798
C01166=1034.798,351.513,-129.999,172.348,45.007,158.797
C01167=1034.790,351.265,-129.961,172.342,45.004,158.795
C01168=1034.783,351.018,-129.923,172.336,45.002,158.794
C01169=1034.775,350.772,-129.886,172.329,45.000,158.793
C01170=1034.767,350.524,-129.847,172.324,44.998,158.792
C01171=1034.759,350.277,-129.810,172.317,44.996,158.791
C01172=1034.747,349.894,-129.751,172.308,44.992,158.789
C01173=1034.736,349.509,-129.692,172.299,44.989,158.787
C01174=1034.724,349.125,-129.634,172.290,44.986,158.786
C01175=1034.712,348.740,-129.575,172.281,44.982,158.784
C01176=1034.704,348.493,-129.538,172.275,44.980,158.783
C01177=1034.696,348.246,-129.500,172.269,44.978,158.782
C01178=1034.688,347.999,-129.463,172.263,44.976,158.781
C01179=1034.681,347.751,-129.425,172.257,44.974,158.780
C01180=1034.673,347.504,-129.388,172.252,44.972,158.778
C01181=1034.665,347.257,-129.351,172.245,44.970,158.777
C01182=1034.658,347.010,-129.313,172.240,44.968,158.776
C01183=1034.650,346.763,-129.276,172.234,44.966,158.775
C01184=1034.643,346.516,-129.239,172.228,44.964,158.774
C01185=1034.635,346.269,-129.202,172.223,44.962,158.773
C01186=1034.627,346.021,-129.164,172.217,44.960,158.772
C01187=1034.619,345.775,-129.127,172.211,44.958,158.771
C01188=1034.612,345.528,-129.090,172.205,44.956,158.770
C01189=1034.605,345.280,-129.052,172.200,44.954,158.769
C01190=1034.597,345.033,-129.016,172.193,44.952,158.768
C01191=1034.590,344.786,-128.978,172.188,44.950,158.767
C01192=1034.582,344.539,-128.941,172.183,44.947,158.766
C01193=1034.574,344.292,-128.904,172.176,44.946,158.765
C01194=1034.566,344.045,-128.867,172.171,44.943,158.764
C01195=1034.560,343.797,-128.830,172.166,44.941,158.763
C01196=1034.552,343.550,-128.793,172.160,44.940,158.762
C01197=1034.544,343.304,-128.756,172.154,44.938,158.761
C01198=1034.537,343.056,-128.719,172.148,44.936,158.760
C01199=1034.529,342.809,-128.683,172.143,44.934,158.759
C01200=1034.521,342.562,-128.645,172.137,44.932,158.758
C01201=1034.514,342.314,-128.609,172.131,44.931,158.757
C01202=1034.506,342.067,-128.571,172.126,44.928,158.756
C01203=1034.499,341.820,-128.535,172.121,44.926,158.755
C01204=1034.492,341.573,-128.498,172.114,44.924,158.753
C01205=1034.484,341.326,-128.462,172.109,44.923,158.753
C01206=1034.477,341.079,-128.425,172.104,44.921,158.752
C01207=1034.470,340.831,-128.388,172.098,44.919,158.751
C01208=1034.462,340.585,-128.351,172.092,44.917,158.750
C01209=1034.454,340.337,-128.315,172.087,44.915,158.749
C01210=1034.446,340.090,-128.279,172.081,44.914,158.748
C01211=1034.439,339.843,-128.241,172.076,44.912,158.747
C01212=1034.431,339.595,-128.205,172.071,44.910,158.746
C01213=1034.424,339.348,-128.169,172.065,44.908,158.745
C01214=1034.416,339.102,-128.132,172.059,44.907,158.744
C01215=1034.409,338.854,-128.096,172.054,44.905,158.743
C01216=1034.402,338.606,-128.059,172.049,44.903,158.742
C01217=1034.394,338.359,-128.023,172.043,44.901,158.741
C01218=1034.386,338.111,-127.987,172.038,44.900,158.740
C01219=1034.379,337.865,-127.950,172.032,44.898,158.739
C01220=1034.371,337.618,-127.914,172.027,44.896,158.738
C01221=1034.364,337.370,-127.877,172.021,44.895,158.737
C01222=1034.357,337.123,-127.841,172.016,44.893,158.736
C01223=1034.350,336.876,-127.805,172.011,44.891,158.735
C01224=1034.342,336.628,-127.769,172.006,44.890,158.734
C01225=1034.334,336.381,-127.732,171.999,44.888,158.733
C01226=1034.328,336.134,-127.696,171.994,44.886,158.733
C01227=1034.320,335.887,-127.660,171.989,44.885,158.732
C01228=1034.308,335.499,-127.603,171.980,44.882,158.730
C01229=1034.297,335.112,-127.546,171.972,44.879,158.729
C01230=1034.286,334.724,-127.489,171.964,44.877,158.727
C01231=1034.274,334.335,-127.433,171.956,44.874,158.726
C01232=1034.266,334.089,-127.398,171.951,44.872,158.725
C01233=1034.259,333.841,-127.361,171.945,44.871,158.724
C01234=1034.251,333.594,-127.325,171.940,44.870,158.723
C01235=1034.244,333.346,-127.290,171.935,44.868,158.722
C01236=1034.237,333.099,-127.254,171.930,44.867,158.722
C01237=1034.229,332.851,-127.218,171.925,44.865,158.721
C01238=1034.222,332.604,-127.182,171.918,44.863,158.720
C01239=1034.215,332.357,-127.146,171.913,44.862,158.719
C01240=1034.208,332.110,-127.110,171.908,44.860,158.718
C01241=1034.200,331.862,-127.075,171.903,44.858,158.717
C01242=1034.193,331.615,-127.039,171.898,44.857,158.716
C01243=1034.185,331.368,-127.003,171.893,44.855,158.715
C01244=1034.178,331.121,-126.968,171.888,44.854,158.714
C01245=1034.170,330.873,-126.932,171.882,44.852,158.714
C01246=1034.163,330.626,-126.897,171.877,44.852,158.713
C01247=1034.156,330.378,-126.861,171.872,44.850,158.712
C01248=1034.149,330.131,-126.826,171.867,44.848,158.711
C01249=1034.141,329.884,-126.789,171.862,44.847,158.710
C01250=1034.135,329.636,-126.754,171.857,44.845,158.709
C01251=1034.127,329.389,-126.718,171.852,44.844,158.709
C01252=1034.120,329.141,-126.683,171.847,44.842,158.708
C01253=1034.112,328.894,-126.647,171.842,44.841,158.707
C01254=1034.106,328.647,-126.611,171.837,44.839,158.706
C01255=1034.099,328.399,-126.576,171.832,44.838,158.705
C01256=1034.090,328.152,-126.541,171.827,44.837,158.704
C01257=1034.084,327.905,-126.506,171.821,44.835,158.703
C01258=1034.076,327.657,-126.471,171.816,44.834,158.703
C01259=1034.069,327.410,-126.436,171.811,44.833,158.702
C01260=1034.061,327.162,-126.401,171.806,44.831,158.701
C01261=1034.054,326.915,-126.365,171.801,44.830,158.700
C01262=1034.046,326.667,-126.330,171.796,44.829,158.700
C01263=1034.039,326.420,-126.295,171.791,44.827,158.699
C01264=1034.031,326.173,-126.260,171.786,44.826,158.698
C01265=1034.024,325.925,-126.225,171.781,44.825,158.697
C01266=1034.016,325.678,-126.190,171.776,44.824,158.696
C01267=1034.010,325.430,-126.155,171.771,44.822,158.696
C01268=1034.002,325.183,-126.120,171.766,44.821,158.695
C01269=1033.995,324.935,-126.085,171.761,44.820,158.694
C01270=1033.987,324.688,-126.050,171.756,44.819,158.693
C01271=1033.980,324.440,-126.015,171.750,44.817,158.692
C01272=1033.972,324.193,-125.980,171.746,44.817,158.692
C01273=1033.966,323.946,-125.945,171.741,44.815,158.691
C01274=1033.957,323.698,-125.910,171.736,44.814,158.690
C01275=1033.951,323.451,-125.875,171.731,44.812,158.689
C01276=1033.944,323.203,-125.841,171.726,44.812,158.689
C01277=1033.936,322.956,-125.807,171.721,44.810,158.688
C01278=1033.929,322.708,-125.771,171.716,44.809,158.687
C01279=1033.921,322.461,-125.737,171.711,44.807,158.686
C01280=1033.914,322.213,-125.702,171.706,44.806,158.686
C01281=1033.907,321.966,-125.667,171.701,44.806,158.685
C01282=1033.900,321.718,-125.633,171.696,44.804,158.684
C01283=1033.892,321.471,-125.598,171.692,44.803,158.683
C01284=1033.881,321.079,-125.543,171.684,44.801,158.682
C01285=1033.870,320.686,-125.488,171.677,44.799,158.681
C01286=1033.859,320.294,-125.433,171.669,44.797,158.680
C01287=1033.848,319.901,-125.378,171.661,44.796,158.679
C01288=1033.840,319.654,-125.344,171.656,44.795,158.678
C01289=1033.833,319.406,-125.308,171.652,44.793,158.677
C01290=1033.826,319.159,-125.275,171.647,44.792,158.676
C01291=1033.819,318.911,-125.239,171.643,44.791,158.676
C01292=1033.811,318.664,-125.205,171.638,44.790,158.675
C01293=1033.804,318.417,-125.171,171.633,44.788,158.674
C01294=1033.797,318.169,-125.136,171.628,44.788,158.673
C01295=1033.790,317.922,-125.102,171.623,44.787,158.673
C01296=1033.783,317.674,-125.067,171.618,44.786,158.672
C01297=1033.776,317.427,-125.033,171.613,44.784,158.671
C01298=1033.769,317.179,-124.998,171.610,44.783,158.671
C01299=1033.762,316.931,-124.964,171.605,44.782,158.670
C01300=1033.755,316.684,-124.930,171.600,44.781,158.669
C01301=1033.748,316.436,-124.895,171.595,44.780,158.669
C01302=1033.741,316.189,-124.861,171.590,44.779,158.668
C01303=1033.734,315.941,-124.826,171.586,44.778,158.667
C01304=1033.727,315.694,-124.792,171.580,44.776,158.666
C01305=1033.720,315.446,-124.757,171.577,44.775,158.666
C01306=1033.713,315.199,-124.724,171.572,44.774,158.665
C01307=1033.707,314.952,-124.690,171.567,44.773,158.664
C01308=1033.700,314.704,-124.655,171.562,44.772,158.664
C01309=1033.693,314.457,-124.621,171.557,44.771,158.663
C01310=1033.686,314.209,-124.587,171.553,44.770,158.662
C01311=1033.679,313.961,-124.553,171.549,44.769,158.662
C01312=1033.671,313.714,-124.518,171.544,44.768,158.661
C01313=1033.665,313.466,-124.484,171.539,44.767,158.660
C01314=1033.658,313.219,-124.450,171.535,44.766,158.660
C01315=1033.651,312.971,-124.417,171.530,44.765,158.659
C01316=1033.645,312.723,-124.382,171.526,44.764,158.658
C01317=1033.637,312.476,-124.348,171.521,44.763,158.657
C01318=1033.631,312.228,-124.313,171.516,44.762,158.657
C01319=1033.624,311.981,-124.280,171.512,44.761,158.656
C01320=1033.617,311.734,-124.246,171.508,44.760,158.655
C01321=1033.610,311.486,-124.212,171.503,44.759,158.655
C01322=1033.603,311.238,-124.178,171.498,44.758,158.654
C01323=1033.595,310.991,-124.144,171.493,44.757,158.653
C01324=1033.588,310.743,-124.111,171.489,44.757,158.653
C01325=1033.582,310.496,-124.077,171.484,44.756,158.652
C01326=1033.574,310.248,-124.043,171.480,44.755,158.652
C01327=1033.567,310.000,-124.010,171.476,44.754,158.651
C01328=1033.560,309.753,-123.977,171.471,44.753,158.650
C01329=1033.552,309.505,-123.943,171.466,44.752,158.650
C01330=1033.546,309.258,-123.910,171.462,44.752,158.649
C01331=1033.539,309.010,-123.876,171.458,44.751,158.648
C01332=1033.531,308.762,-123.843,171.453,44.750,158.648
C01333=1033.524,308.515,-123.810,171.448,44.750,158.647
C01334=1033.516,308.267,-123.776,171.444,44.749,158.647
C01335=1033.510,308.019,-123.743,171.439,44.748,158.646
C01336=1033.503,307.772,-123.709,171.435,44.747,158.645
C01337=1033.495,307.524,-123.676,171.431,44.746,158.645
C01338=1033.489,307.277,-123.643,171.426,44.746,158.644
C01339=1033.482,307.029,-123.609,171.421,44.745,158.644
C01340=1033.470,306.642,-123.557,171.414,44.744,158.643
C01341=1033.459,306.254,-123.505,171.408,44.742,158.642
C01342=1033.448,305.867,-123.453,171.401,44.741,158.641
C01343=1033.438,305.479,-123.401,171.394,44.740,158.640
C01344=1033.430,305.232,-123.368,171.389,44.740,158.639
C01345=1033.423,304.984,-123.335,171.386,44.738,158.639
C01346=1033.416,304.736,-123.301,171.381,44.738,158.638
C01347=1033.409,304.488,-123.268,171.376,44.737,158.637
C01348=1033.402,304.241,-123.235,171.372,44.737,158.637
C01349=1033.395,303.993,-123.202,171.368,44.735,158.636
C01350=1033.389,303.746,-123.169,171.363,44.735,158.636
C01351=1033.382,303.498,-123.135,171.359,44.735,158.635
C01352=1033.374,303.250,-123.103,171.355,44.734,158.635
C01353=1033.367,303.003,-123.069,171.351,44.733,158.634
C01354=1033.360,302.755,-123.036,171.346,44.732,158.633
C01355=1033.354,302.507,-123.004,171.342,44.732,158.633
C01356=1033.346,302.260,-122.970,171.337,44.731,158.632
C01357=1033.340,302.012,-122.938,171.333,44.730,158.632
C01358=1033.333,301.764,-122.905,171.329,44.730,158.631
C01359=1033.326,301.517,-122.871,171.325,44.729,158.631
C01360=1033.319,301.269,-122.839,171.320,44.728,158.630
C01361=1033.313,301.021,-122.806,171.316,44.728,158.630
C01362=1033.305,300.774,-122.772,171.312,44.727,158.629
C01363=1033.299,300.526,-122.739,171.307,44.726,158.628
C01364=1033.291,300.278,-122.707,171.304,44.726,158.628
C01365=1033.285,300.030,-122.674,171.299,44.725,158.627
C01366=1033.278,299.782,-122.641,171.295,44.724,158.627
C01367=1033.271,299.535,-122.608,171.291,44.724,158.626
C01368=1033.265,299.288,-122.575,171.286,44.723,158.625
C01369=1033.258,299.040,-122.542,171.282,44.722,158.625
C01370=1033.251,298.792,-122.509,171.278,44.722,158.624
C01371=1033.244,298.544,-122.477,171.273,44.721,158.624
C01372=1033.237,298.296,-122.444,171.270,44.720,158.623
C01373=1033.231,298.049,-122.411,171.265,44.720,158.623
C01374=1033.224,297.801,-122.378,171.261,44.719,158.622
C01375=1033.217,297.554,-122.345,171.257,44.718,158.622
C01376=1033.211,297.306,-122.313,171.253,44.718,158.621
C01377=1033.204,297.058,-122.280,171.249,44.718,158.621
C01378=1033.197,296.811,-122.247,171.244,44.717,158.620
C01379=1033.190,296.563,-122.215,171.240,44.716,158.619
C01380=1033.184,296.315,-122.182,171.236,44.716,158.619
C01381=1033.177,296.067,-122.149,171.232,44.715,158.618
C01382=1033.170,295.820,-122.117,171.228,44.715,158.618
C01383=1033.163,295.572,-122.084,171.224,44.714,158.617
C01384=1033.157,295.323,-122.052,171.219,44.713,158.617
C01385=1033.150,295.076,-122.019,171.216,44.712,158.616
C01386=1033.143,294.828,-121.986,171.211,44.712,158.616
C01387=1033.137,294.580,-121.954,171.208,44.712,158.615
C01388=1033.130,294.333,-121.921,171.203,44.711,158.615
C01389=1033.123,294.086,-121.889,171.199,44.711,158.614
C01390=1033.116,293.837,-121.857,171.195,44.710,158.614
C01391=1033.109,293.589,-121.825,171.191,44.710,158.613
C01392=1033.102,293.342,-121.793,171.187,44.709,158.613
C01393=1033.096,293.094,-121.759,171.183,44.709,158.612
C01394=1033.089,292.846,-121.728,171.179,44.708,158.612
C01395=1033.083,292.598,-121.695,171.174,44.708,158.611
C01396=1033.072,292.228,-121.647,171.169,44.707,158.611
C01397=1033.061,291.858,-121.600,171.163,44.706,158.610
C01398=1033.051,291.487,-121.552,171.156,44.706,158.609
C01399=1033.041,291.117,-121.504,171.150,44.706,158.608
C01400=1033.035,290.868,-121.472,171.146,44.705,158.608
C01401=1033.027,290.620,-121.439,171.142,44.705,158.607
C01402=1033.020,290.372,-121.408,171.138,44.704,158.607
C01403=1033.013,290.125,-121.376,171.134,44.704,158.606
C01404=1033.007,289.877,-121.344,171.130,44.703,158.606
C01405=1033.000,289.629,-121.311,171.126,44.703,158.605
C01406=1032.993,289.381,-121.280,171.122,44.702,158.605
C01407=1032.986,289.134,-121.248,171.118,44.702,158.605
C01408=1032.980,288.886,-121.215,171.114,44.702,158.604
C01409=1032.973,288.638,-121.184,171.110,44.701,158.604
C01410=1032.966,288.390,-121.152,171.106,44.701,158.603
C01411=1032.959,288.142,-121.120,171.102,44.700,158.603
C01412=1032.952,287.894,-121.088,171.098,44.701,158.602
C01413=1032.945,287.647,-121.057,171.094,44.700,158.602
C01414=1032.939,287.398,-121.025,171.091,44.699,158.601
C01415=1032.932,287.151,-120.992,171.086,44.699,158.601
C01416=1032.925,286.903,-120.961,171.083,44.699,158.600
C01417=1032.919,286.655,-120.929,171.079,44.699,158.600
C01418=1032.912,286.407,-120.898,171.075,44.698,158.599
C01419=1032.904,286.159,-120.866,171.071,44.698,158.599
C01420=1032.898,285.911,-120.834,171.067,44.698,158.599
C01421=1032.891,285.664,-120.803,171.063,44.697,158.598
C01422=1032.884,285.416,-120.771,171.059,44.697,158.598
C01423=1032.877,285.168,-120.740,171.055,44.697,158.597
C01424=1032.871,284.920,-120.708,171.051,44.696,158.597
C01425=1032.864,284.672,-120.677,171.047,44.697,158.596
C01426=1032.857,284.424,-120.646,171.043,44.696,158.596
C01427=1032.850,284.177,-120.613,171.039,44.696,158.596
C01428=1032.843,283.928,-120.582,171.036,44.696,158.595
C01429=1032.836,283.680,-120.550,171.032,44.695,158.595
C01430=1032.830,283.432,-120.519,171.028,44.695,158.594
C01431=1032.823,283.184,-120.487,171.024,44.695,158.594
C01432=1032.816,282.937,-120.456,171.020,44.695,158.593
C01433=1032.809,282.689,-120.425,171.016,44.694,158.593
C01434=1032.802,282.441,-120.394,171.012,44.695,158.593
C01435=1032.795,282.193,-120.362,171.009,44.694,158.592
C01436=1032.788,281.945,-120.331,171.005,44.694,158.592
C01437=1032.782,281.697,-120.300,171.001,44.694,158.591
C01438=1032.775,281.449,-120.269,170.998,44.694,158.591
C01439=1032.769,281.201,-120.237,170.993,44.693,158.591
C01440=1032.762,280.953,-120.206,170.989,44.693,158.590
C01441=1032.755,280.705,-120.174,170.986,44.693,158.590
C01442=1032.748,280.457,-120.143,170.982,44.692,158.589
C01443=1032.742,280.209,-120.111,170.978,44.692,158.589
C01444=1032.735,279.961,-120.080,170.974,44.692,158.588
C01445=1032.728,279.713,-120.049,170.971,44.692,158.588
C01446=1032.722,279.466,-120.018,170.967,44.692,158.588
C01447=1032.715,279.218,-119.987,170.963,44.692,158.587
C01448=1032.708,278.970,-119.956,170.959,44.692,158.587
C01449=1032.701,278.722,-119.924,170.956,44.691,158.586
C01450=1032.695,278.474,-119.893,170.952,44.691,158.586
C01451=1032.688,278.226,-119.862,170.948,44.691,158.586
C01452=1032.679,277.867,-119.818,170.943,44.691,158.585
C01453=1032.668,277.509,-119.772,170.937,44.690,158.584
C01454=1032.659,277.151,-119.727,170.931,44.690,158.584
C01455=1032.649,276.792,-119.683,170.926,44.690,158.583
C01456=1032.642,276.544,-119.652,170.923,44.690,158.583
C01457=1032.635,276.296,-119.621,170.919,44.690,158.583
C01458=1032.630,276.048,-119.590,170.915,44.690,158.582
C01459=1032.622,275.800,-119.560,170.912,44.690,158.582
C01460=1032.615,275.552,-119.528,170.908,44.690,158.582
C01461=1032.609,275.304,-119.497,170.904,44.690,158.581
C01462=1032.602,275.056,-119.467,170.900,44.690,158.581
C01463=1032.595,274.808,-119.436,170.897,44.690,158.580
C01464=1032.588,274.560,-119.404,170.893,44.690,158.580
C01465=1032.582,274.312,-119.375,170.889,44.689,158.580
C01466=1032.575,274.065,-119.343,170.886,44.689,158.579
C01467=1032.569,273.816,-119.313,170.882,44.689,158.579
C01468=1032.562,273.568,-119.282,170.878,44.689,158.579
C01469=1032.555,273.320,-119.251,170.875,44.689,158.578
C01470=1032.548,273.072,-119.221,170.871,44.689,158.578
C01471=1032.542,272.824,-119.190,170.867,44.689,158.577
C01472=1032.534,272.576,-119.160,170.864,44.689,158.577
C01473=1032.528,272.328,-119.129,170.860,44.689,158.577
C01474=1032.521,272.080,-119.098,170.856,44.689,158.576
C01475=1032.515,271.832,-119.068,170.853,44.689,158.576
C01476=1032.508,271.584,-119.037,170.850,44.689,158.576
C01477=1032.501,271.336,-119.006,170.845,44.689,158.575
C01478=1032.494,271.088,-118.975,170.842,44.689,158.575
C01479=1032.488,270.840,-118.946,170.839,44.689,158.575
C01480=1032.481,270.592,-118.915,170.835,44.689,158.574
C01481=1032.474,270.344,-118.884,170.831,44.689,158.574
C01482=1032.468,270.096,-118.853,170.828,44.689,158.574
C01483=1032.461,269.848,-118.824,170.823,44.689,158.573
C01484=1032.455,269.599,-118.793,170.820,44.689,158.573
C01485=1032.447,269.351,-118.763,170.817,44.689,158.573
C01486=1032.441,269.104,-118.732,170.814,44.689,158.572
C01487=1032.434,268.856,-118.702,170.809,44.689,158.572
C01488=1032.427,268.608,-118.672,170.806,44.689,158.572
C01489=1032.421,268.359,-118.641,170.803,44.689,158.571
C01490=1032.414,268.112,-118.611,170.799,44.689,158.571
C01491=1032.408,267.863,-118.580,170.795,44.690,158.571
C01492=1032.400,267.615,-118.550,170.792,44.690,158.570
C01493=1032.394,267.367,-118.520,170.789,44.690,158.570
C01494=1032.387,267.119,-118.490,170.785,44.690,158.570
C01495=1032.380,266.871,-118.460,170.781,44.690,158.569
C01496=1032.374,266.623,-118.429,170.778,44.690,158.569
C01497=1032.367,266.375,-118.399,170.774,44.690,158.569
C01498=1032.360,266.126,-118.369,170.771,44.690,158.568
C01499=1032.354,265.879,-118.339,170.767,44.690,158.568
C01500=1032.347,265.630,-118.309,170.764,44.690,158.568
C01501=1032.340,265.382,-118.278,170.760,44.690,158.567
C01502=1032.333,265.135,-118.249,170.757,44.690,158.567
C01503=1032.326,264.886,-118.219,170.753,44.690,158.567
C01504=1032.320,264.639,-118.188,170.749,44.690,158.566
C01505=1032.313,264.390,-118.158,170.746,44.690,158.566
C01506=1032.306,264.142,-118.129,170.743,44.691,158.566
C01507=1032.300,263.894,-118.099,170.739,44.691,158.565
C01508=1032.290,263.540,-118.056,170.734,44.691,158.565
C01509=1032.281,263.186,-118.013,170.729,44.691,158.565
C01510=1032.271,262.832,-117.970,170.725,44.692,158.564
C01511=1032.262,262.478,-117.928,170.719,44.691,158.564
C01512=1032.255,262.230,-117.897,170.716,44.692,158.563
C01513=1032.248,261.983,-117.868,170.713,44.692,158.563
C01514=1032.242,261.734,-117.837,170.709,44.692,158.563
C01515=1032.236,261.486,-117.808,170.705,44.692,158.563
C01516=1032.229,261.238,-117.778,170.702,44.692,158.562
C01517=1032.222,260.990,-117.748,170.699,44.692,158.562
C01518=1032.215,260.742,-117.719,170.696,44.693,158.562
C01519=1032.207,260.494,-117.689,170.691,44.693,158.561
C01520=1032.201,260.246,-117.660,170.688,44.693,158.561
C01521=1032.194,259.997,-117.630,170.685,44.694,158.561
C01522=1032.188,259.749,-117.601,170.682,44.694,158.561
C01523=1032.181,259.501,-117.571,170.677,44.694,158.560
C01524=1032.174,259.253,-117.542,170.674,44.695,158.560
C01525=1032.167,259.005,-117.512,170.671,44.695,158.560
C01526=1032.160,258.757,-117.483,170.668,44.695,158.560
C01527=1032.153,258.509,-117.453,170.665,44.696,158.559
C01528=1032.146,258.260,-117.424,170.661,44.696,158.559
C01529=1032.140,258.012,-117.394,170.657,44.696,158.559
C01530=1032.133,257.763,-117.364,170.654,44.696,158.559
C01531=1032.126,257.516,-117.335,170.651,44.696,158.558
C01532=1032.119,257.267,-117.306,170.648,44.697,158.558
C01533=1032.112,257.019,-117.277,170.644,44.697,158.558
C01534=1032.105,256.771,-117.247,170.640,44.697,158.557
C01535=1032.099,256.523,-117.218,170.637,44.698,158.557
C01536=1032.092,256.274,-117.188,170.634,44.698,158.557
C01537=1032.085,256.027,-117.159,170.631,44.698,158.557
C01538=1032.079,255.779,-117.130,170.628,44.699,158.556
C01539=1032.072,255.530,-117.101,170.623,44.699,158.556
C01540=1032.065,255.282,-117.071,170.620,44.700,158.556
C01541=1032.058,255.034,-117.042,170.617,44.700,158.556
C01542=1032.052,254.785,-117.012,170.614,44.700,158.555
C01543=1032.045,254.537,-116.982,170.611,44.700,158.555
C01544=1032.038,254.289,-116.954,170.607,44.700,158.555
C01545=1032.032,254.041,-116.925,170.603,44.701,158.555
C01546=1032.024,253.793,-116.895,170.600,44.701,158.554
C01547=1032.018,253.545,-116.866,170.597,44.702,158.554
C01548=1032.011,253.296,-116.836,170.594,44.702,158.554
C01549=1032.005,253.048,-116.807,170.591,44.702,158.554
C01550=1031.998,252.800,-116.779,170.588,44.702,158.553
C01551=1031.991,252.552,-116.749,170.584,44.703,158.553
C01552=1031.985,252.304,-116.720,170.581,44.703,158.553
C01553=1031.978,252.055,-116.690,170.577,44.703,158.553
C01554=1031.972,251.807,-116.661,170.574,44.704,158.552
C01555=1031.965,251.559,-116.633,170.571,44.704,158.552
C01556=1031.958,251.310,-116.603,170.568,44.705,158.552
C01557=1031.951,251.063,-116.574,170.564,44.705,158.552
C01558=1031.945,250.815,-116.545,170.561,44.705,158.551
C01559=1031.938,250.566,-116.515,170.558,44.705,158.551
C01560=1031.931,250.318,-116.487,170.555,44.705,158.551
C01561=1031.925,250.070,-116.458,170.552,44.706,158.551
C01562=1031.919,249.822,-116.429,170.548,44.706,158.550
C01563=1031.912,249.573,-116.399,170.545,44.707,158.550
C01564=1031.902,249.217,-116.357,170.540,44.707,158.550
C01565=1031.893,248.863,-116.316,170.536,44.707,158.549
C01566=1031.884,248.507,-116.275,170.531,44.708,158.549
C01567=1031.874,248.152,-116.233,170.526,44.709,158.549
C01568=1031.867,247.904,-116.204,170.523,44.709,158.549
C01569=1031.861,247.656,-116.175,170.520,44.709,158.548
C01570=1031.855,247.408,-116.146,170.517,44.709,158.548
C01571=1031.848,247.159,-116.117,170.514,44.710,158.548
C01572=1031.842,246.911,-116.088,170.511,44.711,158.548
C01573=1031.835,246.663,-116.059,170.507,44.711,158.547
C01574=1031.828,246.415,-116.030,170.504,44.711,158.547
C01575=1031.822,246.166,-116.001,170.501,44.711,158.547
C01576=1031.815,245.918,-115.972,170.498,44.712,158.547
C01577=1031.809,245.670,-115.943,170.495,44.712,158.547
C01578=1031.802,245.422,-115.914,170.492,44.713,158.546
C01579=1031.796,245.173,-115.886,170.488,44.713,158.546
C01580=1031.790,244.925,-115.857,170.485,44.713,158.546
C01581=1031.783,244.676,-115.828,170.482,44.713,158.546
C01582=1031.776,244.428,-115.799,170.479,44.714,158.545
C01583=1031.770,244.180,-115.770,170.475,44.715,158.545
C01584=1031.763,243.932,-115.742,170.472,44.715,158.545
C01585=1031.757,243.684,-115.713,170.469,44.715,158.545
C01586=1031.751,243.435,-115.684,170.466,44.716,158.545
C01587=1031.743,243.187,-115.655,170.462,44.716,158.544
C01588=1031.737,242.938,-115.627,170.459,44.717,158.544
C01589=1031.730,242.690,-115.599,170.456,44.717,158.544
C01590=1031.724,242.442,-115.570,170.453,44.717,158.544
C01591=1031.717,242.194,-115.542,170.450,44.718,158.544
C01592=1031.711,241.946,-115.513,170.447,44.719,158.543
C01593=1031.703,241.697,-115.484,170.444,44.719,158.543
C01594=1031.697,241.448,-115.456,170.441,44.719,158.543
C01595=1031.690,241.201,-115.427,170.438,44.720,158.543
C01596=1031.684,240.952,-115.398,170.435,44.721,158.543
C01597=1031.677,240.704,-115.370,170.431,44.721,158.542
C01598=1031.671,240.456,-115.341,170.428,44.721,158.542
C01599=1031.665,240.207,-115.314,170.425,44.722,158.542
C01600=1031.657,239.959,-115.285,170.422,44.723,158.542
C01601=1031.651,239.710,-115.257,170.419,44.723,158.542
C01602=1031.644,239.462,-115.228,170.416,44.723,158.541
C01603=1031.637,239.214,-115.200,170.413,44.724,158.541
C01604=1031.630,238.966,-115.172,170.410,44.725,158.541
C01605=1031.624,238.717,-115.144,170.407,44.725,158.541
C01606=1031.617,238.469,-115.115,170.404,44.726,158.541
C01607=1031.611,238.221,-115.087,170.400,44.726,158.540
C01608=1031.603,237.972,-115.059,170.397,44.727,158.540
C01609=1031.597,237.724,-115.030,170.394,44.727,158.540
C01610=1031.591,237.475,-115.003,170.391,44.728,158.540
C01611=1031.584,237.227,-114.974,170.388,44.728,158.540
C01612=1031.577,236.979,-114.946,170.385,44.729,158.540
C01613=1031.571,236.731,-114.917,170.382,44.730,158.540
C01614=1031.564,236.482,-114.890,170.379,44.730,158.539
C01615=1031.557,236.234,-114.862,170.376,44.730,158.539
C01616=1031.550,235.986,-114.833,170.373,44.731,158.539
C01617=1031.544,235.738,-114.806,170.370,44.732,158.539
C01618=1031.538,235.489,-114.777,170.367,44.732,158.539
C01619=1031.531,235.241,-114.750,170.364,44.733,158.538
C01620=1031.521,234.880,-114.709,170.360,44.734,158.538
C01621=1031.511,234.518,-114.668,170.356,44.735,158.538
C01622=1031.501,234.157,-114.627,170.351,44.736,158.538
C01623=1031.491,233.795,-114.587,170.346,44.736,158.537
C01624=1031.485,233.547,-114.558,170.343,44.737,158.537
C01625=1031.478,233.299,-114.530,170.340,44.737,158.537
C01626=1031.472,233.050,-114.502,170.337,44.738,158.537
C01627=1031.465,232.802,-114.474,170.334,44.739,158.537
C01628=1031.459,232.554,-114.447,170.331,44.739,158.537
C01629=1031.452,232.306,-114.419,170.328,44.740,158.536
C01630=1031.446,232.058,-114.390,170.325,44.741,158.536
C01631=1031.439,231.809,-114.363,170.322,44.741,158.536
C01632=1031.433,231.561,-114.335,170.319,44.742,158.536
C01633=1031.426,231.312,-114.307,170.316,44.743,158.536
C01634=1031.419,231.064,-114.279,170.314,44.743,158.536
C01635=1031.413,230.815,-114.252,170.311,44.744,158.536
C01636=1031.406,230.567,-114.224,170.308,44.744,158.535
C01637=1031.399,230.319,-114.195,170.305,44.745,158.535
C01638=1031.392,230.071,-114.168,170.302,44.746,158.535
C01639=1031.386,229.822,-114.140,170.299,44.746,158.535
C01640=1031.379,229.574,-114.112,170.296,44.747,158.535
C01641=1031.372,229.325,-114.085,170.293,44.747,158.535
C01642=1031.366,229.077,-114.057,170.290,44.748,158.534
C01643=1031.359,228.829,-114.029,170.287,44.749,158.534
C01644=1031.352,228.580,-114.001,170.284,44.749,158.534
C01645=1031.346,228.332,-113.974,170.281,44.750,158.534
C01646=1031.339,228.084,-113.946,170.277,44.751,158.534
C01647=1031.333,227.836,-113.919,170.275,44.751,158.534
C01648=1031.326,227.586,-113.892,170.272,44.752,158.534
C01649=1031.320,227.338,-113.864,170.269,44.752,158.533
C01650=1031.313,227.090,-113.836,170.266,44.753,158.533
C01651=1031.306,226.841,-113.808,170.264,44.754,158.533
C01652=1031.299,226.593,-113.781,170.261,44.755,158.533
C01653=1031.292,226.345,-113.753,170.257,44.756,158.533
C01654=1031.286,226.096,-113.726,170.254,44.756,158.533
C01655=1031.279,225.847,-113.699,170.251,44.757,158.533
C01656=1031.273,225.599,-113.671,170.248,44.758,158.532
C01657=1031.266,225.351,-113.644,170.246,44.759,158.533
C01658=1031.259,225.103,-113.616,170.243,44.760,158.532
C01659=1031.253,224.854,-113.589,170.239,44.760,158.532
C01660=1031.246,224.605,-113.562,170.237,44.761,158.532
C01661=1031.239,224.357,-113.535,170.234,44.761,158.532
C01662=1031.232,224.109,-113.507,170.231,44.762,158.532
C01663=1031.226,223.860,-113.480,170.229,44.763,158.532
C01664=1031.219,223.612,-113.453,170.226,44.764,158.532
C01665=1031.213,223.363,-113.425,170.223,44.764,158.531
C01666=1031.205,223.115,-113.398,170.219,44.765,158.531
C01667=1031.199,222.866,-113.371,170.216,44.766,158.531
C01668=1031.192,222.618,-113.343,170.213,44.766,158.531
C01669=1031.186,222.370,-113.316,170.212,44.768,158.531
C01670=1031.179,222.121,-113.289,170.209,44.768,158.531
C01671=1031.172,221.873,-113.261,170.206,44.769,158.531
C01672=1031.166,221.624,-113.234,170.203,44.769,158.531
C01673=1031.159,221.375,-113.207,170.199,44.770,158.530
C01674=1031.153,221.128,-113.180,170.197,44.771,158.530
C01675=1031.146,220.880,-113.152,170.194,44.772,158.530
C01676=1031.136,220.511,-113.112,170.190,44.773,158.530
C01677=1031.126,220.141,-113.071,170.186,44.774,158.530
C01678=1031.117,219.772,-113.031,170.182,44.775,158.530
C01679=1031.107,219.404,-112.990,170.177,44.776,158.530
C01680=1031.100,219.155,-112.963,170.175,44.777,158.529
C01681=1031.093,218.908,-112.937,170.172,44.778,158.529
C01682=1031.087,218.659,-112.910,170.169,44.779,158.529
C01683=1031.080,218.410,-112.883,170.166,44.779,158.529
C01684=1031.073,218.161,-112.855,170.163,44.781,158.529
C01685=1031.067,217.913,-112.829,170.160,44.781,158.529
C01686=1031.060,217.665,-112.802,170.157,44.782,158.529
C01687=1031.053,217.416,-112.775,170.155,44.783,158.529
C01688=1031.046,217.168,-112.748,170.152,44.784,158.529
C01689=1031.040,216.920,-112.721,170.149,44.784,158.529
C01690=1031.033,216.671,-112.694,170.146,44.786,158.529
C01691=1031.026,216.422,-112.667,170.143,44.786,158.528
C01692=1031.020,216.173,-112.640,170.140,44.787,158.528
C01693=1031.013,215.925,-112.614,170.137,44.788,158.528
C01694=1031.006,215.677,-112.587,170.135,44.789,158.528
C01695=1030.999,215.428,-112.560,170.133,44.790,158.528
C01696=1030.993,215.180,-112.533,170.130,44.791,158.528
C01697=1030.986,214.932,-112.506,170.127,44.791,158.528
C01698=1030.979,214.683,-112.480,170.124,44.792,158.528
C01699=1030.973,214.434,-112.453,170.121,44.793,158.528
C01700=1030.966,214.186,-112.426,170.119,44.794,158.528
C01701=1030.959,213.937,-112.399,170.116,44.795,158.528
C01702=1030.952,213.689,-112.373,170.113,44.796,158.527
C01703=1030.946,213.441,-112.345,170.110,44.796,158.527
C01704=1030.939,213.192,-112.319,170.107,44.797,158.527
C01705=1030.933,212.944,-112.292,170.105,44.798,158.527
C01706=1030.926,212.695,-112.266,170.102,44.799,158.527
C01707=1030.919,212.447,-112.238,170.099,44.800,158.527
C01708=1030.913,212.198,-112.212,170.096,44.800,158.527
C01709=1030.907,211.949,-112.185,170.093,44.802,158.527
C01710=1030.899,211.701,-112.159,170.091,44.802,158.527
C01711=1030.894,211.452,-112.132,170.088,44.803,158.527
C01712=1030.886,211.204,-112.105,170.086,44.804,158.527
C01713=1030.880,210.956,-112.079,170.082,44.805,158.526
C01714=1030.873,210.707,-112.052,170.080,44.806,158.526
C01715=1030.866,210.458,-112.025,170.078,44.806,158.526
C01716=1030.860,210.210,-111.999,170.075,44.808,158.526
C01717=1030.853,209.961,-111.972,170.072,44.808,158.526
C01718=1030.846,209.712,-111.946,170.069,44.810,158.526
C01719=1030.839,209.465,-111.919,170.066,44.810,158.526
C01720=1030.832,209.216,-111.893,170.064,44.811,158.526
C01721=1030.827,208.968,-111.866,170.061,44.812,158.526
C01722=1030.819,208.719,-111.840,170.058,44.813,158.526
C01723=1030.812,208.470,-111.813,170.055,44.814,158.526
C01724=1030.807,208.222,-111.787,170.053,44.814,158.526
C01725=1030.799,207.973,-111.760,170.051,44.816,158.526
C01726=1030.793,207.725,-111.734,170.048,44.817,158.526
C01727=1030.786,207.477,-111.708,170.045,44.818,158.525
C01728=1030.779,207.228,-111.682,170.042,44.819,158.525
C01729=1030.773,206.979,-111.655,170.040,44.819,158.525
C01730=1030.766,206.731,-111.628,170.037,44.821,158.525
C01731=1030.759,206.483,-111.602,170.034,44.821,158.525
C01732=1030.750,206.119,-111.564,170.030,44.823,158.525
C01733=1030.739,205.756,-111.526,170.026,44.824,158.525
C01734=1030.729,205.394,-111.487,170.023,44.826,158.525
C01735=1030.720,205.031,-111.450,170.019,44.827,158.525
C01736=1030.694,203.981,-111.344,169.664,44.724,158.469
C01737=1030.688,203.733,-111.319,169.660,44.725,158.469
C01738=1030.683,203.484,-111.295,169.657,44.727,158.469
C01739=1030.676,203.235,-111.269,169.653,44.729,158.469
C01740=1030.670,202.988,-111.245,169.650,44.730,158.469
C01741=1030.664,202.738,-111.220,169.646,44.732,158.469
C01742=1030.658,202.490,-111.195,169.643,44.734,158.469
C01743=1030.652,202.240,-111.170,169.639,44.735,158.469
C01744=1030.646,201.992,-111.145,169.635,44.737,158.469
C01745=1030.641,201.743,-111.121,169.632,44.739,158.469
C01746=1030.634,201.495,-111.096,169.628,44.740,158.469
C01747=1030.628,201.246,-111.072,169.624,44.743,158.469
C01748=1030.622,200.998,-111.046,169.620,44.744,158.469
C01749=1030.616,200.748,-111.022,169.617,44.746,158.469
C01750=1030.611,200.500,-110.997,169.613,44.748,158.469
C01751=1030.605,200.251,-110.972,169.610,44.750,158.469
C01752=1030.598,200.002,-110.948,169.606,44.751,158.469
C01753=1030.592,199.754,-110.923,169.602,44.753,158.469
C01754=1030.586,199.505,-110.899,169.599,44.755,158.469
C01755=1030.579,199.256,-110.875,169.596,44.757,158.469
C01756=1030.574,199.008,-110.850,169.592,44.759,158.469
C01757=1030.567,198.759,-110.826,169.588,44.761,158.469
C01758=1030.561,198.510,-110.801,169.585,44.763,158.469
C01759=1030.555,198.262,-110.778,169.581,44.765,158.469
C01760=1030.549,198.013,-110.752,169.577,44.766,158.469
C01761=1030.542,197.764,-110.728,169.574,44.769,158.469
C01762=1030.537,197.515,-110.704,169.570,44.770,158.469
C01763=1030.530,197.266,-110.680,169.567,44.772,158.469
C01764=1030.524,197.017,-110.656,169.563,44.774,158.469
C01765=1030.518,196.769,-110.631,169.559,44.776,158.469
C01766=1030.512,196.520,-110.607,169.556,44.778,158.470
C01767=1030.506,196.272,-110.583,169.553,44.780,158.470
C01768=1030.500,196.023,-110.558,169.549,44.781,158.470
C01769=1030.493,195.774,-110.534,169.546,44.784,158.470
C01770=1030.488,195.525,-110.510,169.542,44.786,158.470
C01771=1030.481,195.277,-110.485,169.538,44.787,158.470
C01772=1030.476,195.028,-110.461,169.535,44.789,158.470
C01773=1030.469,194.779,-110.437,169.531,44.792,158.470
C01774=1030.464,194.530,-110.413,169.527,44.793,158.470
C01775=1030.457,194.282,-110.389,169.525,44.795,158.470
C01776=1030.451,194.032,-110.364,169.521,44.797,158.470
C01777=1030.445,193.784,-110.340,169.517,44.799,158.470
